bogBasketRotCtClockWiseMoveAllow.AppScalingDivisor :=1;
bogBasketRotCtClockWiseMoveAllow.AppScalingMultiplier :=1;
bogBasketRotCtClockWiseMoveAllow.AppScalingOffset :=0;
bogBasketRotCtClockWiseMoveAllow.AppUnit :="";
bogBasketRotCtClockWiseMoveAllow.CanDefault :=0;
bogBasketRotCtClockWiseMoveAllow.CanInit :=0;
bogBasketRotCtClockWiseMoveAllow.CanMax :=1;
bogBasketRotCtClockWiseMoveAllow.CanMin :=0;
bogBasketRotCtClockWiseMoveAllow.CanUnit :="";
bogBasketRotCtClockWiseMoveAllow.Description :="Basket Rotation Counter Clockwise Move Allowed";
bogBasketRotCtClockWiseMoveAllow.ErrorReaction := eErrorReaction.ERSIG_DFLT;
bogBasketRotCtClockWiseMoveAllow.ReceiverAdress :=1;
bogBasketRotCtClockWiseMoveAllow.ToolScalingDivisor :=1;
bogBasketRotCtClockWiseMoveAllow.ToolScalingMultiplier :=1;
bogBasketRotCtClockWiseMoveAllow.ToolScalingOffset :=0;
bogBasketRotCtClockWiseMoveAllow.ToolUnit :="";

bogBasketRotClockWiseMoveAllow.AppScalingDivisor :=1;
bogBasketRotClockWiseMoveAllow.AppScalingMultiplier :=1;
bogBasketRotClockWiseMoveAllow.AppScalingOffset :=0;
bogBasketRotClockWiseMoveAllow.AppUnit :="";
bogBasketRotClockWiseMoveAllow.CanDefault :=0;
bogBasketRotClockWiseMoveAllow.CanInit :=0;
bogBasketRotClockWiseMoveAllow.CanMax :=1;
bogBasketRotClockWiseMoveAllow.CanMin :=0;
bogBasketRotClockWiseMoveAllow.CanUnit :="";
bogBasketRotClockWiseMoveAllow.Description :="Basket Rotation Clockwise Move Allowed";
bogBasketRotClockWiseMoveAllow.ErrorReaction := eErrorReaction.ERSIG_DFLT;
bogBasketRotClockWiseMoveAllow.ReceiverAdress :=1;
bogBasketRotClockWiseMoveAllow.ToolScalingDivisor :=1;
bogBasketRotClockWiseMoveAllow.ToolScalingMultiplier :=1;
bogBasketRotClockWiseMoveAllow.ToolScalingOffset :=0;
bogBasketRotClockWiseMoveAllow.ToolUnit :="";

bogBasketInclinMoveUpAllow.AppScalingDivisor :=1;
bogBasketInclinMoveUpAllow.AppScalingMultiplier :=1;
bogBasketInclinMoveUpAllow.AppScalingOffset :=0;
bogBasketInclinMoveUpAllow.AppUnit :="";
bogBasketInclinMoveUpAllow.CanDefault :=0;
bogBasketInclinMoveUpAllow.CanInit :=0;
bogBasketInclinMoveUpAllow.CanMax :=1;
bogBasketInclinMoveUpAllow.CanMin :=0;
bogBasketInclinMoveUpAllow.CanUnit :="";
bogBasketInclinMoveUpAllow.Description :="Basket Inclinaison Move Up Allowed";
bogBasketInclinMoveUpAllow.ErrorReaction := eErrorReaction.ERSIG_DFLT;
bogBasketInclinMoveUpAllow.ReceiverAdress :=1;
bogBasketInclinMoveUpAllow.ToolScalingDivisor :=1;
bogBasketInclinMoveUpAllow.ToolScalingMultiplier :=1;
bogBasketInclinMoveUpAllow.ToolScalingOffset :=0;
bogBasketInclinMoveUpAllow.ToolUnit :="";

bogBasketInclinMoveDownAllow.AppScalingDivisor :=1;
bogBasketInclinMoveDownAllow.AppScalingMultiplier :=1;
bogBasketInclinMoveDownAllow.AppScalingOffset :=0;
bogBasketInclinMoveDownAllow.AppUnit :="";
bogBasketInclinMoveDownAllow.CanDefault :=0;
bogBasketInclinMoveDownAllow.CanInit :=0;
bogBasketInclinMoveDownAllow.CanMax :=1;
bogBasketInclinMoveDownAllow.CanMin :=0;
bogBasketInclinMoveDownAllow.CanUnit :="";
bogBasketInclinMoveDownAllow.Description :="Basket Inclinaison Move Down Allowed";
bogBasketInclinMoveDownAllow.ErrorReaction := eErrorReaction.ERSIG_DFLT;
bogBasketInclinMoveDownAllow.ReceiverAdress :=1;
bogBasketInclinMoveDownAllow.ToolScalingDivisor :=1;
bogBasketInclinMoveDownAllow.ToolScalingMultiplier :=1;
bogBasketInclinMoveDownAllow.ToolScalingOffset :=0;
bogBasketInclinMoveDownAllow.ToolUnit :="";

bogVehiculeDefault.AppScalingDivisor :=1;
bogVehiculeDefault.AppScalingMultiplier :=1;
bogVehiculeDefault.AppScalingOffset :=0;
bogVehiculeDefault.AppUnit :="";
bogVehiculeDefault.CanDefault :=0;
bogVehiculeDefault.CanInit :=0;
bogVehiculeDefault.CanMax :=1;
bogVehiculeDefault.CanMin :=0;
bogVehiculeDefault.CanUnit :="";
bogVehiculeDefault.Description :="Vehicule in Default (A12)";
bogVehiculeDefault.ErrorReaction := eErrorReaction.ERSIG_DFLT;
bogVehiculeDefault.ReceiverAdress :=1;
bogVehiculeDefault.ToolScalingDivisor :=1;
bogVehiculeDefault.ToolScalingMultiplier :=1;
bogVehiculeDefault.ToolScalingOffset :=0;
bogVehiculeDefault.ToolUnit :="";

bogTelescopeOutputPossible.AppScalingDivisor :=1;
bogTelescopeOutputPossible.AppScalingMultiplier :=1;
bogTelescopeOutputPossible.AppScalingOffset :=0;
bogTelescopeOutputPossible.AppUnit :="";
bogTelescopeOutputPossible.CanDefault :=0;
bogTelescopeOutputPossible.CanInit :=0;
bogTelescopeOutputPossible.CanMax :=1;
bogTelescopeOutputPossible.CanMin :=0;
bogTelescopeOutputPossible.CanUnit :="";
bogTelescopeOutputPossible.Description :="Telescope output possible (A48)";
bogTelescopeOutputPossible.ErrorReaction := eErrorReaction.ERSIG_DFLT;
bogTelescopeOutputPossible.ReceiverAdress :=1;
bogTelescopeOutputPossible.ToolScalingDivisor :=1;
bogTelescopeOutputPossible.ToolScalingMultiplier :=1;
bogTelescopeOutputPossible.ToolScalingOffset :=0;
bogTelescopeOutputPossible.ToolUnit :="";

bogTelescopeWinderFault.AppScalingDivisor :=1;
bogTelescopeWinderFault.AppScalingMultiplier :=1;
bogTelescopeWinderFault.AppScalingOffset :=0;
bogTelescopeWinderFault.AppUnit :="";
bogTelescopeWinderFault.CanDefault :=0;
bogTelescopeWinderFault.CanInit :=0;
bogTelescopeWinderFault.CanMax :=1;
bogTelescopeWinderFault.CanMin :=0;
bogTelescopeWinderFault.CanUnit :="";
bogTelescopeWinderFault.Description :="Telescope Winder Fault (A17)";
bogTelescopeWinderFault.ErrorReaction := eErrorReaction.ERSIG_DFLT;
bogTelescopeWinderFault.ReceiverAdress :=1;
bogTelescopeWinderFault.ToolScalingDivisor :=1;
bogTelescopeWinderFault.ToolScalingMultiplier :=1;
bogTelescopeWinderFault.ToolScalingOffset :=0;
bogTelescopeWinderFault.ToolUnit :="";

bogNacellePostSelector.AppScalingDivisor :=1;
bogNacellePostSelector.AppScalingMultiplier :=1;
bogNacellePostSelector.AppScalingOffset :=0;
bogNacellePostSelector.AppUnit :="";
bogNacellePostSelector.CanDefault :=0;
bogNacellePostSelector.CanInit :=0;
bogNacellePostSelector.CanMax :=1;
bogNacellePostSelector.CanMin :=0;
bogNacellePostSelector.CanUnit :="";
bogNacellePostSelector.Description :="Nacelle post selector";
bogNacellePostSelector.ErrorReaction := eErrorReaction.ERSIG_DFLT;
bogNacellePostSelector.ReceiverAdress :=1;
bogNacellePostSelector.ToolScalingDivisor :=1;
bogNacellePostSelector.ToolScalingMultiplier :=1;
bogNacellePostSelector.ToolScalingOffset :=0;
bogNacellePostSelector.ToolUnit :="";

bogSTOP_On_Off.AppScalingDivisor :=1;
bogSTOP_On_Off.AppScalingMultiplier :=1;
bogSTOP_On_Off.AppScalingOffset :=0;
bogSTOP_On_Off.AppUnit :="";
bogSTOP_On_Off.CanDefault :=0;
bogSTOP_On_Off.CanInit :=0;
bogSTOP_On_Off.CanMax :=1;
bogSTOP_On_Off.CanMin :=0;
bogSTOP_On_Off.CanUnit :="";
bogSTOP_On_Off.Description :="STOP Status";
bogSTOP_On_Off.ErrorReaction := eErrorReaction.ERSIG_DFLT;
bogSTOP_On_Off.ReceiverAdress :=1;
bogSTOP_On_Off.ToolScalingDivisor :=1;
bogSTOP_On_Off.ToolScalingMultiplier :=1;
bogSTOP_On_Off.ToolScalingOffset :=0;
bogSTOP_On_Off.ToolUnit :="";

bogSafeManSystem.AppScalingDivisor :=1;
bogSafeManSystem.AppScalingMultiplier :=1;
bogSafeManSystem.AppScalingOffset :=0;
bogSafeManSystem.AppUnit :="";
bogSafeManSystem.CanDefault :=0;
bogSafeManSystem.CanInit :=0;
bogSafeManSystem.CanMax :=1;
bogSafeManSystem.CanMin :=0;
bogSafeManSystem.CanUnit :="";
bogSafeManSystem.Description :="SafeManSystem (A5)";
bogSafeManSystem.ErrorReaction := eErrorReaction.ERSIG_DFLT;
bogSafeManSystem.ReceiverAdress :=1;
bogSafeManSystem.ToolScalingDivisor :=1;
bogSafeManSystem.ToolScalingMultiplier :=1;
bogSafeManSystem.ToolScalingOffset :=0;
bogSafeManSystem.ToolUnit :="";

bogHighSpeedAllow.AppScalingDivisor :=1;
bogHighSpeedAllow.AppScalingMultiplier :=1;
bogHighSpeedAllow.AppScalingOffset :=0;
bogHighSpeedAllow.AppUnit :="";
bogHighSpeedAllow.CanDefault :=0;
bogHighSpeedAllow.CanInit :=0;
bogHighSpeedAllow.CanMax :=1;
bogHighSpeedAllow.CanMin :=0;
bogHighSpeedAllow.CanUnit :="";
bogHighSpeedAllow.Description :="High Speed Allow (A19)";
bogHighSpeedAllow.ErrorReaction := eErrorReaction.ERSIG_DFLT;
bogHighSpeedAllow.ReceiverAdress :=1;
bogHighSpeedAllow.ToolScalingDivisor :=1;
bogHighSpeedAllow.ToolScalingMultiplier :=1;
bogHighSpeedAllow.ToolScalingOffset :=0;
bogHighSpeedAllow.ToolUnit :="";

bogAutomatiqueStop.AppScalingDivisor :=1;
bogAutomatiqueStop.AppScalingMultiplier :=1;
bogAutomatiqueStop.AppScalingOffset :=0;
bogAutomatiqueStop.AppUnit :="";
bogAutomatiqueStop.CanDefault :=0;
bogAutomatiqueStop.CanInit :=0;
bogAutomatiqueStop.CanMax :=1;
bogAutomatiqueStop.CanMin :=0;
bogAutomatiqueStop.CanUnit :="";
bogAutomatiqueStop.Description :="Automatique Stop or function mismatch (A20)";
bogAutomatiqueStop.ErrorReaction := eErrorReaction.ERSIG_DFLT;
bogAutomatiqueStop.ReceiverAdress :=1;
bogAutomatiqueStop.ToolScalingDivisor :=1;
bogAutomatiqueStop.ToolScalingMultiplier :=1;
bogAutomatiqueStop.ToolScalingOffset :=0;
bogAutomatiqueStop.ToolUnit :="";

bogLowSpeedByFault.AppScalingDivisor :=1;
bogLowSpeedByFault.AppScalingMultiplier :=1;
bogLowSpeedByFault.AppScalingOffset :=0;
bogLowSpeedByFault.AppUnit :="";
bogLowSpeedByFault.CanDefault :=0;
bogLowSpeedByFault.CanInit :=0;
bogLowSpeedByFault.CanMax :=1;
bogLowSpeedByFault.CanMin :=0;
bogLowSpeedByFault.CanUnit :="";
bogLowSpeedByFault.Description :="Low Speed by fault (A46)";
bogLowSpeedByFault.ErrorReaction := eErrorReaction.ERSIG_DFLT;
bogLowSpeedByFault.ReceiverAdress :=1;
bogLowSpeedByFault.ToolScalingDivisor :=1;
bogLowSpeedByFault.ToolScalingMultiplier :=1;
bogLowSpeedByFault.ToolScalingOffset :=0;
bogLowSpeedByFault.ToolUnit :="";

bogMeasuringMastFault.AppScalingDivisor :=1;
bogMeasuringMastFault.AppScalingMultiplier :=1;
bogMeasuringMastFault.AppScalingOffset :=0;
bogMeasuringMastFault.AppUnit :="";
bogMeasuringMastFault.CanDefault :=0;
bogMeasuringMastFault.CanInit :=0;
bogMeasuringMastFault.CanMax :=1;
bogMeasuringMastFault.CanMin :=0;
bogMeasuringMastFault.CanUnit :="";
bogMeasuringMastFault.Description :="Measuring Mast in Fault (A8)";
bogMeasuringMastFault.ErrorReaction := eErrorReaction.ERSIG_DFLT;
bogMeasuringMastFault.ReceiverAdress :=1;
bogMeasuringMastFault.ToolScalingDivisor :=1;
bogMeasuringMastFault.ToolScalingMultiplier :=1;
bogMeasuringMastFault.ToolScalingOffset :=0;
bogMeasuringMastFault.ToolUnit :="";

bogMeasuringMatOption.AppScalingDivisor :=1;
bogMeasuringMatOption.AppScalingMultiplier :=1;
bogMeasuringMatOption.AppScalingOffset :=0;
bogMeasuringMatOption.AppUnit :="";
bogMeasuringMatOption.CanDefault :=0;
bogMeasuringMatOption.CanInit :=0;
bogMeasuringMatOption.CanMax :=1;
bogMeasuringMatOption.CanMin :=0;
bogMeasuringMatOption.CanUnit :="";
bogMeasuringMatOption.Description :="Measuring mast option";
bogMeasuringMatOption.ErrorReaction := eErrorReaction.ERSIG_DFLT;
bogMeasuringMatOption.ReceiverAdress :=1;
bogMeasuringMatOption.ToolScalingDivisor :=1;
bogMeasuringMatOption.ToolScalingMultiplier :=1;
bogMeasuringMatOption.ToolScalingOffset :=0;
bogMeasuringMatOption.ToolUnit :="";

bogBasketAccessLocked.AppScalingDivisor :=1;
bogBasketAccessLocked.AppScalingMultiplier :=1;
bogBasketAccessLocked.AppScalingOffset :=0;
bogBasketAccessLocked.AppUnit :="";
bogBasketAccessLocked.CanDefault :=0;
bogBasketAccessLocked.CanInit :=0;
bogBasketAccessLocked.CanMax :=1;
bogBasketAccessLocked.CanMin :=0;
bogBasketAccessLocked.CanUnit :="";
bogBasketAccessLocked.Description :="Basket access locked";
bogBasketAccessLocked.ErrorReaction := eErrorReaction.ERSIG_DFLT;
bogBasketAccessLocked.ReceiverAdress :=1;
bogBasketAccessLocked.ToolScalingDivisor :=1;
bogBasketAccessLocked.ToolScalingMultiplier :=1;
bogBasketAccessLocked.ToolScalingOffset :=0;
bogBasketAccessLocked.ToolUnit :="";

bogFilterOverloadNoActive.AppScalingDivisor :=1;
bogFilterOverloadNoActive.AppScalingMultiplier :=1;
bogFilterOverloadNoActive.AppScalingOffset :=0;
bogFilterOverloadNoActive.AppUnit :="";
bogFilterOverloadNoActive.CanDefault :=0;
bogFilterOverloadNoActive.CanInit :=0;
bogFilterOverloadNoActive.CanMax :=1;
bogFilterOverloadNoActive.CanMin :=0;
bogFilterOverloadNoActive.CanUnit :="";
bogFilterOverloadNoActive.Description :="new signal";
bogFilterOverloadNoActive.ErrorReaction := eErrorReaction.ERSIG_DFLT;
bogFilterOverloadNoActive.ReceiverAdress :=1;
bogFilterOverloadNoActive.ToolScalingDivisor :=1;
bogFilterOverloadNoActive.ToolScalingMultiplier :=1;
bogFilterOverloadNoActive.ToolScalingOffset :=0;
bogFilterOverloadNoActive.ToolUnit :="";

bogAnticlockwiseBasketSlew.AppScalingDivisor :=1;
bogAnticlockwiseBasketSlew.AppScalingMultiplier :=1;
bogAnticlockwiseBasketSlew.AppScalingOffset :=0;
bogAnticlockwiseBasketSlew.AppUnit :="";
bogAnticlockwiseBasketSlew.CanDefault :=0;
bogAnticlockwiseBasketSlew.CanInit :=0;
bogAnticlockwiseBasketSlew.CanMax :=1;
bogAnticlockwiseBasketSlew.CanMin :=0;
bogAnticlockwiseBasketSlew.CanUnit :="";
bogAnticlockwiseBasketSlew.Description :="EV113 Anticlockwise Basket Slew";
bogAnticlockwiseBasketSlew.ErrorReaction := eErrorReaction.ERSIG_DFLT;
bogAnticlockwiseBasketSlew.ReceiverAdress :=1;
bogAnticlockwiseBasketSlew.ToolScalingDivisor :=1;
bogAnticlockwiseBasketSlew.ToolScalingMultiplier :=1;
bogAnticlockwiseBasketSlew.ToolScalingOffset :=0;
bogAnticlockwiseBasketSlew.ToolUnit :="";

bogClockwiseBasketSlew.AppScalingDivisor :=1;
bogClockwiseBasketSlew.AppScalingMultiplier :=1;
bogClockwiseBasketSlew.AppScalingOffset :=0;
bogClockwiseBasketSlew.AppUnit :="";
bogClockwiseBasketSlew.CanDefault :=0;
bogClockwiseBasketSlew.CanInit :=0;
bogClockwiseBasketSlew.CanMax :=1;
bogClockwiseBasketSlew.CanMin :=0;
bogClockwiseBasketSlew.CanUnit :="";
bogClockwiseBasketSlew.Description :="EV112 Anticlockwise Basket Slew";
bogClockwiseBasketSlew.ErrorReaction := eErrorReaction.ERSIG_DFLT;
bogClockwiseBasketSlew.ReceiverAdress :=1;
bogClockwiseBasketSlew.ToolScalingDivisor :=1;
bogClockwiseBasketSlew.ToolScalingMultiplier :=1;
bogClockwiseBasketSlew.ToolScalingOffset :=0;
bogClockwiseBasketSlew.ToolUnit :="";

bogFlashLightForced.AppScalingDivisor :=1;
bogFlashLightForced.AppScalingMultiplier :=1;
bogFlashLightForced.AppScalingOffset :=0;
bogFlashLightForced.AppUnit :="";
bogFlashLightForced.CanDefault :=0;
bogFlashLightForced.CanInit :=0;
bogFlashLightForced.CanMax :=1;
bogFlashLightForced.CanMin :=0;
bogFlashLightForced.CanUnit :="";
bogFlashLightForced.Description :="Flash Light Forced";
bogFlashLightForced.ErrorReaction := eErrorReaction.ERSIG_DFLT;
bogFlashLightForced.ReceiverAdress :=1;
bogFlashLightForced.ToolScalingDivisor :=1;
bogFlashLightForced.ToolScalingMultiplier :=1;
bogFlashLightForced.ToolScalingOffset :=0;
bogFlashLightForced.ToolUnit :="";

bogBasketAccessLockOption.AppScalingDivisor :=1;
bogBasketAccessLockOption.AppScalingMultiplier :=1;
bogBasketAccessLockOption.AppScalingOffset :=0;
bogBasketAccessLockOption.AppUnit :="";
bogBasketAccessLockOption.CanDefault :=0;
bogBasketAccessLockOption.CanInit :=0;
bogBasketAccessLockOption.CanMax :=1;
bogBasketAccessLockOption.CanMin :=0;
bogBasketAccessLockOption.CanUnit :="";
bogBasketAccessLockOption.Description :="Basket Lock Option";
bogBasketAccessLockOption.ErrorReaction := eErrorReaction.ERSIG_DFLT;
bogBasketAccessLockOption.ReceiverAdress :=1;
bogBasketAccessLockOption.ToolScalingDivisor :=1;
bogBasketAccessLockOption.ToolScalingMultiplier :=1;
bogBasketAccessLockOption.ToolScalingOffset :=0;
bogBasketAccessLockOption.ToolUnit :="";

bogBasketLateralStopOption.AppScalingDivisor :=1;
bogBasketLateralStopOption.AppScalingMultiplier :=1;
bogBasketLateralStopOption.AppScalingOffset :=0;
bogBasketLateralStopOption.AppUnit :="";
bogBasketLateralStopOption.CanDefault :=0;
bogBasketLateralStopOption.CanInit :=0;
bogBasketLateralStopOption.CanMax :=1;
bogBasketLateralStopOption.CanMin :=0;
bogBasketLateralStopOption.CanUnit :="";
bogBasketLateralStopOption.Description :="Basket lateral stop option";
bogBasketLateralStopOption.ErrorReaction := eErrorReaction.ERSIG_DFLT;
bogBasketLateralStopOption.ReceiverAdress :=1;
bogBasketLateralStopOption.ToolScalingDivisor :=1;
bogBasketLateralStopOption.ToolScalingMultiplier :=1;
bogBasketLateralStopOption.ToolScalingOffset :=0;
bogBasketLateralStopOption.ToolUnit :="";

bogBasketStepClosed.AppScalingDivisor :=1;
bogBasketStepClosed.AppScalingMultiplier :=1;
bogBasketStepClosed.AppScalingOffset :=0;
bogBasketStepClosed.AppUnit :="";
bogBasketStepClosed.CanDefault :=0;
bogBasketStepClosed.CanInit :=0;
bogBasketStepClosed.CanMax :=1;
bogBasketStepClosed.CanMin :=0;
bogBasketStepClosed.CanUnit :="";
bogBasketStepClosed.Description :="Basket step closed";
bogBasketStepClosed.ErrorReaction := eErrorReaction.ERSIG_DFLT;
bogBasketStepClosed.ReceiverAdress :=1;
bogBasketStepClosed.ToolScalingDivisor :=1;
bogBasketStepClosed.ToolScalingMultiplier :=1;
bogBasketStepClosed.ToolScalingOffset :=0;
bogBasketStepClosed.ToolUnit :="";

bogSystemFault.AppScalingDivisor :=1;
bogSystemFault.AppScalingMultiplier :=1;
bogSystemFault.AppScalingOffset :=0;
bogSystemFault.AppUnit :="";
bogSystemFault.CanDefault :=0;
bogSystemFault.CanInit :=0;
bogSystemFault.CanMax :=1;
bogSystemFault.CanMin :=0;
bogSystemFault.CanUnit :="";
bogSystemFault.Description :="System Fault";
bogSystemFault.ErrorReaction := eErrorReaction.ERSIG_DFLT;
bogSystemFault.ReceiverAdress :=1;
bogSystemFault.ToolScalingDivisor :=1;
bogSystemFault.ToolScalingMultiplier :=1;
bogSystemFault.ToolScalingOffset :=0;
bogSystemFault.ToolUnit :="";

bogTrans1PressureSensorFault.AppScalingDivisor :=1;
bogTrans1PressureSensorFault.AppScalingMultiplier :=1;
bogTrans1PressureSensorFault.AppScalingOffset :=0;
bogTrans1PressureSensorFault.AppUnit :="";
bogTrans1PressureSensorFault.CanDefault :=0;
bogTrans1PressureSensorFault.CanInit :=0;
bogTrans1PressureSensorFault.CanMax :=1;
bogTrans1PressureSensorFault.CanMin :=0;
bogTrans1PressureSensorFault.CanUnit :="";
bogTrans1PressureSensorFault.Description :="Fault pressure transmission 1";
bogTrans1PressureSensorFault.ErrorReaction := eErrorReaction.ERSIG_DFLT;
bogTrans1PressureSensorFault.ReceiverAdress :=1;
bogTrans1PressureSensorFault.ToolScalingDivisor :=1;
bogTrans1PressureSensorFault.ToolScalingMultiplier :=1;
bogTrans1PressureSensorFault.ToolScalingOffset :=0;
bogTrans1PressureSensorFault.ToolUnit :="";

bogTrans2PressureSensorFault.AppScalingDivisor :=1;
bogTrans2PressureSensorFault.AppScalingMultiplier :=1;
bogTrans2PressureSensorFault.AppScalingOffset :=0;
bogTrans2PressureSensorFault.AppUnit :="";
bogTrans2PressureSensorFault.CanDefault :=0;
bogTrans2PressureSensorFault.CanInit :=0;
bogTrans2PressureSensorFault.CanMax :=1;
bogTrans2PressureSensorFault.CanMin :=0;
bogTrans2PressureSensorFault.CanUnit :="";
bogTrans2PressureSensorFault.Description :="Fault pressure transmission 2";
bogTrans2PressureSensorFault.ErrorReaction := eErrorReaction.ERSIG_DFLT;
bogTrans2PressureSensorFault.ReceiverAdress :=1;
bogTrans2PressureSensorFault.ToolScalingDivisor :=1;
bogTrans2PressureSensorFault.ToolScalingMultiplier :=1;
bogTrans2PressureSensorFault.ToolScalingOffset :=0;
bogTrans2PressureSensorFault.ToolUnit :="";

bogOverloadSecurity.AppScalingDivisor :=1;
bogOverloadSecurity.AppScalingMultiplier :=1;
bogOverloadSecurity.AppScalingOffset :=0;
bogOverloadSecurity.AppUnit :="";
bogOverloadSecurity.CanDefault :=0;
bogOverloadSecurity.CanInit :=0;
bogOverloadSecurity.CanMax :=1;
bogOverloadSecurity.CanMin :=0;
bogOverloadSecurity.CanUnit :="";
bogOverloadSecurity.Description :="Basket overload";
bogOverloadSecurity.ErrorReaction := eErrorReaction.ERSIG_DFLT;
bogOverloadSecurity.ReceiverAdress :=1;
bogOverloadSecurity.ToolScalingDivisor :=1;
bogOverloadSecurity.ToolScalingMultiplier :=1;
bogOverloadSecurity.ToolScalingOffset :=0;
bogOverloadSecurity.ToolUnit :="";

bogDeltaArmJoysCenteredTeles.AppScalingDivisor :=1;
bogDeltaArmJoysCenteredTeles.AppScalingMultiplier :=1;
bogDeltaArmJoysCenteredTeles.AppScalingOffset :=0;
bogDeltaArmJoysCenteredTeles.AppUnit :="";
bogDeltaArmJoysCenteredTeles.CanDefault :=0;
bogDeltaArmJoysCenteredTeles.CanInit :=0;
bogDeltaArmJoysCenteredTeles.CanMax :=1;
bogDeltaArmJoysCenteredTeles.CanMin :=0;
bogDeltaArmJoysCenteredTeles.CanUnit :="";
bogDeltaArmJoysCenteredTeles.Description :="Delta and Telescope Joystick centered";
bogDeltaArmJoysCenteredTeles.ErrorReaction := eErrorReaction.ERSIG_DFLT;
bogDeltaArmJoysCenteredTeles.ReceiverAdress :=1;
bogDeltaArmJoysCenteredTeles.ToolScalingDivisor :=1;
bogDeltaArmJoysCenteredTeles.ToolScalingMultiplier :=1;
bogDeltaArmJoysCenteredTeles.ToolScalingOffset :=0;
bogDeltaArmJoysCenteredTeles.ToolUnit :="";

bogArrowJoystickCenteredTurret.AppScalingDivisor :=1;
bogArrowJoystickCenteredTurret.AppScalingMultiplier :=1;
bogArrowJoystickCenteredTurret.AppScalingOffset :=0;
bogArrowJoystickCenteredTurret.AppUnit :="";
bogArrowJoystickCenteredTurret.CanDefault :=0;
bogArrowJoystickCenteredTurret.CanInit :=0;
bogArrowJoystickCenteredTurret.CanMax :=1;
bogArrowJoystickCenteredTurret.CanMin :=0;
bogArrowJoystickCenteredTurret.CanUnit :="";
bogArrowJoystickCenteredTurret.Description :="Arrow and Turret Joystick centered";
bogArrowJoystickCenteredTurret.ErrorReaction := eErrorReaction.ERSIG_DFLT;
bogArrowJoystickCenteredTurret.ReceiverAdress :=1;
bogArrowJoystickCenteredTurret.ToolScalingDivisor :=1;
bogArrowJoystickCenteredTurret.ToolScalingMultiplier :=1;
bogArrowJoystickCenteredTurret.ToolScalingOffset :=0;
bogArrowJoystickCenteredTurret.ToolUnit :="";

bogDeltaArmMoveUp.AppScalingDivisor :=1;
bogDeltaArmMoveUp.AppScalingMultiplier :=1;
bogDeltaArmMoveUp.AppScalingOffset :=0;
bogDeltaArmMoveUp.AppUnit :="";
bogDeltaArmMoveUp.CanDefault :=0;
bogDeltaArmMoveUp.CanInit :=0;
bogDeltaArmMoveUp.CanMax :=1;
bogDeltaArmMoveUp.CanMin :=0;
bogDeltaArmMoveUp.CanUnit :="";
bogDeltaArmMoveUp.Description :="Delta Arm Move Up";
bogDeltaArmMoveUp.ErrorReaction := eErrorReaction.ERSIG_DFLT;
bogDeltaArmMoveUp.ReceiverAdress :=1;
bogDeltaArmMoveUp.ToolScalingDivisor :=1;
bogDeltaArmMoveUp.ToolScalingMultiplier :=1;
bogDeltaArmMoveUp.ToolScalingOffset :=0;
bogDeltaArmMoveUp.ToolUnit :="";

bogDeltaArmMoveDown.AppScalingDivisor :=1;
bogDeltaArmMoveDown.AppScalingMultiplier :=1;
bogDeltaArmMoveDown.AppScalingOffset :=0;
bogDeltaArmMoveDown.AppUnit :="";
bogDeltaArmMoveDown.CanDefault :=0;
bogDeltaArmMoveDown.CanInit :=0;
bogDeltaArmMoveDown.CanMax :=1;
bogDeltaArmMoveDown.CanMin :=0;
bogDeltaArmMoveDown.CanUnit :="";
bogDeltaArmMoveDown.Description :="Delta Arm Move Down";
bogDeltaArmMoveDown.ErrorReaction := eErrorReaction.ERSIG_DFLT;
bogDeltaArmMoveDown.ReceiverAdress :=1;
bogDeltaArmMoveDown.ToolScalingDivisor :=1;
bogDeltaArmMoveDown.ToolScalingMultiplier :=1;
bogDeltaArmMoveDown.ToolScalingOffset :=0;
bogDeltaArmMoveDown.ToolUnit :="";

bogArrowArmMoveUp.AppScalingDivisor :=1;
bogArrowArmMoveUp.AppScalingMultiplier :=1;
bogArrowArmMoveUp.AppScalingOffset :=0;
bogArrowArmMoveUp.AppUnit :="";
bogArrowArmMoveUp.CanDefault :=0;
bogArrowArmMoveUp.CanInit :=0;
bogArrowArmMoveUp.CanMax :=1;
bogArrowArmMoveUp.CanMin :=0;
bogArrowArmMoveUp.CanUnit :="";
bogArrowArmMoveUp.Description :="Arrow Arm Move Up";
bogArrowArmMoveUp.ErrorReaction := eErrorReaction.ERSIG_DFLT;
bogArrowArmMoveUp.ReceiverAdress :=1;
bogArrowArmMoveUp.ToolScalingDivisor :=1;
bogArrowArmMoveUp.ToolScalingMultiplier :=1;
bogArrowArmMoveUp.ToolScalingOffset :=0;
bogArrowArmMoveUp.ToolUnit :="";

bogArrowArmMoveDown.AppScalingDivisor :=1;
bogArrowArmMoveDown.AppScalingMultiplier :=1;
bogArrowArmMoveDown.AppScalingOffset :=0;
bogArrowArmMoveDown.AppUnit :="";
bogArrowArmMoveDown.CanDefault :=0;
bogArrowArmMoveDown.CanInit :=0;
bogArrowArmMoveDown.CanMax :=1;
bogArrowArmMoveDown.CanMin :=0;
bogArrowArmMoveDown.CanUnit :="";
bogArrowArmMoveDown.Description :="Arrow Arm Move Down";
bogArrowArmMoveDown.ErrorReaction := eErrorReaction.ERSIG_DFLT;
bogArrowArmMoveDown.ReceiverAdress :=1;
bogArrowArmMoveDown.ToolScalingDivisor :=1;
bogArrowArmMoveDown.ToolScalingMultiplier :=1;
bogArrowArmMoveDown.ToolScalingOffset :=0;
bogArrowArmMoveDown.ToolUnit :="";

bogTelescopeMoveOut.AppScalingDivisor :=1;
bogTelescopeMoveOut.AppScalingMultiplier :=1;
bogTelescopeMoveOut.AppScalingOffset :=0;
bogTelescopeMoveOut.AppUnit :="";
bogTelescopeMoveOut.CanDefault :=0;
bogTelescopeMoveOut.CanInit :=0;
bogTelescopeMoveOut.CanMax :=1;
bogTelescopeMoveOut.CanMin :=0;
bogTelescopeMoveOut.CanUnit :="";
bogTelescopeMoveOut.Description :="Telescope Move Out";
bogTelescopeMoveOut.ErrorReaction := eErrorReaction.ERSIG_DFLT;
bogTelescopeMoveOut.ReceiverAdress :=1;
bogTelescopeMoveOut.ToolScalingDivisor :=1;
bogTelescopeMoveOut.ToolScalingMultiplier :=1;
bogTelescopeMoveOut.ToolScalingOffset :=0;
bogTelescopeMoveOut.ToolUnit :="";

bogTelescopeMoveIn.AppScalingDivisor :=1;
bogTelescopeMoveIn.AppScalingMultiplier :=1;
bogTelescopeMoveIn.AppScalingOffset :=0;
bogTelescopeMoveIn.AppUnit :="";
bogTelescopeMoveIn.CanDefault :=0;
bogTelescopeMoveIn.CanInit :=0;
bogTelescopeMoveIn.CanMax :=1;
bogTelescopeMoveIn.CanMin :=0;
bogTelescopeMoveIn.CanUnit :="";
bogTelescopeMoveIn.Description :="Telescope Move In";
bogTelescopeMoveIn.ErrorReaction := eErrorReaction.ERSIG_DFLT;
bogTelescopeMoveIn.ReceiverAdress :=1;
bogTelescopeMoveIn.ToolScalingDivisor :=1;
bogTelescopeMoveIn.ToolScalingMultiplier :=1;
bogTelescopeMoveIn.ToolScalingOffset :=0;
bogTelescopeMoveIn.ToolUnit :="";

bogTurretCounterClockWiseMove.AppScalingDivisor :=1;
bogTurretCounterClockWiseMove.AppScalingMultiplier :=1;
bogTurretCounterClockWiseMove.AppScalingOffset :=0;
bogTurretCounterClockWiseMove.AppUnit :="";
bogTurretCounterClockWiseMove.CanDefault :=0;
bogTurretCounterClockWiseMove.CanInit :=0;
bogTurretCounterClockWiseMove.CanMax :=1;
bogTurretCounterClockWiseMove.CanMin :=0;
bogTurretCounterClockWiseMove.CanUnit :="";
bogTurretCounterClockWiseMove.Description :="Turret Counter Clockwise Move";
bogTurretCounterClockWiseMove.ErrorReaction := eErrorReaction.ERSIG_DFLT;
bogTurretCounterClockWiseMove.ReceiverAdress :=1;
bogTurretCounterClockWiseMove.ToolScalingDivisor :=1;
bogTurretCounterClockWiseMove.ToolScalingMultiplier :=1;
bogTurretCounterClockWiseMove.ToolScalingOffset :=0;
bogTurretCounterClockWiseMove.ToolUnit :="";

bogTurretClockWiseMove.AppScalingDivisor :=1;
bogTurretClockWiseMove.AppScalingMultiplier :=1;
bogTurretClockWiseMove.AppScalingOffset :=0;
bogTurretClockWiseMove.AppUnit :="";
bogTurretClockWiseMove.CanDefault :=0;
bogTurretClockWiseMove.CanInit :=0;
bogTurretClockWiseMove.CanMax :=1;
bogTurretClockWiseMove.CanMin :=0;
bogTurretClockWiseMove.CanUnit :="";
bogTurretClockWiseMove.Description :="Turret Clockwise Move";
bogTurretClockWiseMove.ErrorReaction := eErrorReaction.ERSIG_DFLT;
bogTurretClockWiseMove.ReceiverAdress :=1;
bogTurretClockWiseMove.ToolScalingDivisor :=1;
bogTurretClockWiseMove.ToolScalingMultiplier :=1;
bogTurretClockWiseMove.ToolScalingOffset :=0;
bogTurretClockWiseMove.ToolUnit :="";

bogTurretEncoderFault.AppScalingDivisor :=1;
bogTurretEncoderFault.AppScalingMultiplier :=1;
bogTurretEncoderFault.AppScalingOffset :=0;
bogTurretEncoderFault.AppUnit :="";
bogTurretEncoderFault.CanDefault :=0;
bogTurretEncoderFault.CanInit :=0;
bogTurretEncoderFault.CanMax :=1;
bogTurretEncoderFault.CanMin :=0;
bogTurretEncoderFault.CanUnit :="";
bogTurretEncoderFault.Description :="Turret Encoder Fault";
bogTurretEncoderFault.ErrorReaction := eErrorReaction.ERSIG_DFLT;
bogTurretEncoderFault.ReceiverAdress :=1;
bogTurretEncoderFault.ToolScalingDivisor :=1;
bogTurretEncoderFault.ToolScalingMultiplier :=1;
bogTurretEncoderFault.ToolScalingOffset :=0;
bogTurretEncoderFault.ToolUnit :="";

bogGeneratorOption.AppScalingDivisor :=1;
bogGeneratorOption.AppScalingMultiplier :=1;
bogGeneratorOption.AppScalingOffset :=0;
bogGeneratorOption.AppUnit :="";
bogGeneratorOption.CanDefault :=0;
bogGeneratorOption.CanInit :=0;
bogGeneratorOption.CanMax :=1;
bogGeneratorOption.CanMin :=0;
bogGeneratorOption.CanUnit :="";
bogGeneratorOption.Description :="Generator Option";
bogGeneratorOption.ErrorReaction := eErrorReaction.ERSIG_DFLT;
bogGeneratorOption.ReceiverAdress :=1;
bogGeneratorOption.ToolScalingDivisor :=1;
bogGeneratorOption.ToolScalingMultiplier :=1;
bogGeneratorOption.ToolScalingOffset :=0;
bogGeneratorOption.ToolUnit :="";

bogGeneratorActive.AppScalingDivisor :=1;
bogGeneratorActive.AppScalingMultiplier :=1;
bogGeneratorActive.AppScalingOffset :=0;
bogGeneratorActive.AppUnit :="";
bogGeneratorActive.CanDefault :=0;
bogGeneratorActive.CanInit :=0;
bogGeneratorActive.CanMax :=1;
bogGeneratorActive.CanMin :=0;
bogGeneratorActive.CanUnit :="";
bogGeneratorActive.Description :="Generator Active";
bogGeneratorActive.ErrorReaction := eErrorReaction.ERSIG_DFLT;
bogGeneratorActive.ReceiverAdress :=1;
bogGeneratorActive.ToolScalingDivisor :=1;
bogGeneratorActive.ToolScalingMultiplier :=1;
bogGeneratorActive.ToolScalingOffset :=0;
bogGeneratorActive.ToolUnit :="";


                
END_METHOD
END_FUNCTION_BLOCK

FUNCTION_BLOCK Msg2C1SendToEvision7MessageClass EXTENDS CanReceiveMessageClass
  VAR_INPUT
    u8gFuel : UInt8CanSignalClass;
    u16gBattery_Voltage : UInt16CanSignalClass;
    u8gTrainTransmissionPressure : UInt8CanSignalClass;
    i16gBypassPressureSensorValue : Int16CanSignalClass;
    Counter : UInt32CanSignalClass;
  END_VAR

            
          

METHOD SetData
  VAR_INPUT
    CanMsgPointer : POINTER TO CanMessageClass;
  END_VAR
                  IF IsValidPointer(canMsgPointer,'SetData') THEN
	SUPER^.SetData(CanMsgPointer);
	//Set the new data
	u8gFuel.Value := canMsgPointer^.GetUint8(0);
	u16gBattery_Voltage.Value := canMsgPointer^.GetUint16(8);
	u8gTrainTransmissionPressure.Value := canMsgPointer^.GetUint8(24);
	i16gBypassPressureSensorValue.Value := canMsgPointer^.GetInt16(32);
	//And increase the counter
	Counter.Value := CanMsgPointer^.Counter.Value;
END_IF

                
END_METHOD

PROPERTY u8gFuelRawValue : USINT
GET
                    IF u8gFuel.AppScalingMultiplier = 0 THEN
	_MatchLog^.Error("Get u8gFuelRawValue", "Division by Zero!");
	RETURN;
End_IF

u8gFuelRawValue := TO_USINT((u8gFuel.Value - u8gFuel.AppScalingOffset) * u8gFuel.AppScalingDivisor / u8gFuel.AppScalingMultiplier);

                  
END_GET
END_PROPERTY

PROPERTY u16gBattery_VoltageRawValue : UINT
GET
                    IF u16gBattery_Voltage.AppScalingMultiplier = 0 THEN
	_MatchLog^.Error("Get u16gBattery_VoltageRawValue", "Division by Zero!");
	RETURN;
End_IF

u16gBattery_VoltageRawValue := TO_UINT((u16gBattery_Voltage.Value - u16gBattery_Voltage.AppScalingOffset) * u16gBattery_Voltage.AppScalingDivisor / u16gBattery_Voltage.AppScalingMultiplier);

                  
END_GET
END_PROPERTY

PROPERTY u8gTrainTransmissionPressureRawValue : USINT
GET
                    IF u8gTrainTransmissionPressure.AppScalingMultiplier = 0 THEN
	_MatchLog^.Error("Get u8gTrainTransmissionPressureRawValue", "Division by Zero!");
	RETURN;
End_IF

u8gTrainTransmissionPressureRawValue := TO_USINT((u8gTrainTransmissionPressure.Value - u8gTrainTransmissionPressure.AppScalingOffset) * u8gTrainTransmissionPressure.AppScalingDivisor / u8gTrainTransmissionPressure.AppScalingMultiplier);

                  
END_GET
END_PROPERTY

PROPERTY i16gBypassPressureSensorValueRawValue : INT
GET
                    IF i16gBypassPressureSensorValue.AppScalingMultiplier = 0 THEN
	_MatchLog^.Error("Get i16gBypassPressureSensorValueRawValue", "Division by Zero!");
	RETURN;
End_IF

i16gBypassPressureSensorValueRawValue := TO_INT((i16gBypassPressureSensorValue.Value - i16gBypassPressureSensorValue.AppScalingOffset) * i16gBypassPressureSensorValue.AppScalingDivisor / i16gBypassPressureSensorValue.AppScalingMultiplier);

                  
END_GET
END_PROPERTY

PROPERTY u8gFuelToolValue : USINT
GET
                    IF u8gFuel.ToolScalingDivisor = 0 OR u8gFuel.AppScalingMultiplier = 0 THEN
	_MatchLog^.Error("Get u8gFuelToolValue", "Division by Zero!");
	RETURN;
END_IF

u8gFuelToolValue := TO_USINT(((u8gFuel.Value - u8gFuel.AppScalingOffset) * u8gFuel.AppScalingDivisor / u8gFuel.AppScalingMultiplier * u8gFuel.ToolScalingMultiplier / u8gFuel.ToolScalingDivisor) + u8gFuel.ToolScalingOffset);

                  
END_GET
END_PROPERTY

PROPERTY u16gBattery_VoltageToolValue : UINT
GET
                    IF u16gBattery_Voltage.ToolScalingDivisor = 0 OR u16gBattery_Voltage.AppScalingMultiplier = 0 THEN
	_MatchLog^.Error("Get u16gBattery_VoltageToolValue", "Division by Zero!");
	RETURN;
END_IF

u16gBattery_VoltageToolValue := TO_UINT(((u16gBattery_Voltage.Value - u16gBattery_Voltage.AppScalingOffset) * u16gBattery_Voltage.AppScalingDivisor / u16gBattery_Voltage.AppScalingMultiplier * u16gBattery_Voltage.ToolScalingMultiplier / u16gBattery_Voltage.ToolScalingDivisor) + u16gBattery_Voltage.ToolScalingOffset);

                  
END_GET
END_PROPERTY

PROPERTY u8gTrainTransmissionPressureToolValue : USINT
GET
                    IF u8gTrainTransmissionPressure.ToolScalingDivisor = 0 OR u8gTrainTransmissionPressure.AppScalingMultiplier = 0 THEN
	_MatchLog^.Error("Get u8gTrainTransmissionPressureToolValue", "Division by Zero!");
	RETURN;
END_IF

u8gTrainTransmissionPressureToolValue := TO_USINT(((u8gTrainTransmissionPressure.Value - u8gTrainTransmissionPressure.AppScalingOffset) * u8gTrainTransmissionPressure.AppScalingDivisor / u8gTrainTransmissionPressure.AppScalingMultiplier * u8gTrainTransmissionPressure.ToolScalingMultiplier / u8gTrainTransmissionPressure.ToolScalingDivisor) + u8gTrainTransmissionPressure.ToolScalingOffset);

                  
END_GET
END_PROPERTY

PROPERTY i16gBypassPressureSensorValueToolValue : INT
GET
                    IF i16gBypassPressureSensorValue.ToolScalingDivisor = 0 OR i16gBypassPressureSensorValue.AppScalingMultiplier = 0 THEN
	_MatchLog^.Error("Get i16gBypassPressureSensorValueToolValue", "Division by Zero!");
	RETURN;
END_IF

i16gBypassPressureSensorValueToolValue := TO_INT(((i16gBypassPressureSensorValue.Value - i16gBypassPressureSensorValue.AppScalingOffset) * i16gBypassPressureSensorValue.AppScalingDivisor / i16gBypassPressureSensorValue.AppScalingMultiplier * i16gBypassPressureSensorValue.ToolScalingMultiplier / i16gBypassPressureSensorValue.ToolScalingDivisor) + i16gBypassPressureSensorValue.ToolScalingOffset);

                  
END_GET
END_PROPERTY

METHOD InitializeCanSignals
                  u8gFuel.AppScalingDivisor :=1;
u8gFuel.AppScalingMultiplier :=1;
u8gFuel.AppScalingOffset :=0;
u8gFuel.AppUnit :="";
u8gFuel.CanDefault :=0;
u8gFuel.CanInit :=0;
u8gFuel.CanMax :=255;
u8gFuel.CanMin :=0;
u8gFuel.CanUnit :="";
u8gFuel.Description :="new signal";
u8gFuel.ErrorReaction := eErrorReaction.ERSIG_DFLT;
u8gFuel.ReceiverAdress :=1;
u8gFuel.ToolScalingDivisor :=1;
u8gFuel.ToolScalingMultiplier :=1;
u8gFuel.ToolScalingOffset :=0;
u8gFuel.ToolUnit :="";

u16gBattery_Voltage.AppScalingDivisor :=1;
u16gBattery_Voltage.AppScalingMultiplier :=1;
u16gBattery_Voltage.AppScalingOffset :=0;
u16gBattery_Voltage.AppUnit :="";
u16gBattery_Voltage.CanDefault :=0;
u16gBattery_Voltage.CanInit :=0;
u16gBattery_Voltage.CanMax :=65535;
u16gBattery_Voltage.CanMin :=0;
u16gBattery_Voltage.CanUnit :="";
u16gBattery_Voltage.Description :="new signal";
u16gBattery_Voltage.ErrorReaction := eErrorReaction.ERSIG_DFLT;
u16gBattery_Voltage.ReceiverAdress :=1;
u16gBattery_Voltage.ToolScalingDivisor :=1;
u16gBattery_Voltage.ToolScalingMultiplier :=1;
u16gBattery_Voltage.ToolScalingOffset :=0;
u16gBattery_Voltage.ToolUnit :="";

u8gTrainTransmissionPressure.AppScalingDivisor :=1;
u8gTrainTransmissionPressure.AppScalingMultiplier :=1;
u8gTrainTransmissionPressure.AppScalingOffset :=0;
u8gTrainTransmissionPressure.AppUnit :="";
u8gTrainTransmissionPressure.CanDefault :=0;
u8gTrainTransmissionPressure.CanInit :=0;
u8gTrainTransmissionPressure.CanMax :=255;
u8gTrainTransmissionPressure.CanMin :=0;
u8gTrainTransmissionPressure.CanUnit :="";
u8gTrainTransmissionPressure.Description :="new signal";
u8gTrainTransmissionPressure.ErrorReaction := eErrorReaction.ERSIG_DFLT;
u8gTrainTransmissionPressure.ReceiverAdress :=1;
u8gTrainTransmissionPressure.ToolScalingDivisor :=1;
u8gTrainTransmissionPressure.ToolScalingMultiplier :=1;
u8gTrainTransmissionPressure.ToolScalingOffset :=0;
u8gTrainTransmissionPressure.ToolUnit :="";

i16gBypassPressureSensorValue.AppScalingDivisor :=1;
i16gBypassPressureSensorValue.AppScalingMultiplier :=1;
i16gBypassPressureSensorValue.AppScalingOffset :=0;
i16gBypassPressureSensorValue.AppUnit :="";
i16gBypassPressureSensorValue.CanDefault :=0;
i16gBypassPressureSensorValue.CanInit :=0;
i16gBypassPressureSensorValue.CanMax :=VBasic.LibConst.I16_MAX;
i16gBypassPressureSensorValue.CanMin :=VBasic.LibConst.I16_MIN;
i16gBypassPressureSensorValue.CanUnit :="";
i16gBypassPressureSensorValue.Description :="new signal";
i16gBypassPressureSensorValue.ErrorReaction := eErrorReaction.ERSIG_DFLT;
i16gBypassPressureSensorValue.ReceiverAdress :=1;
i16gBypassPressureSensorValue.ToolScalingDivisor :=1;
i16gBypassPressureSensorValue.ToolScalingMultiplier :=1;
i16gBypassPressureSensorValue.ToolScalingOffset :=0;
i16gBypassPressureSensorValue.ToolUnit :="";


                
END_METHOD
END_FUNCTION_BLOCK

FUNCTION_BLOCK Msg3C1SendToEvision7MessageClass EXTENDS CanReceiveMessageClass
  VAR_INPUT
    u32MinValueEncodeurMast : UInt32CanSignalClass;
    u32MaxValueEncodeurMast : UInt32CanSignalClass;
    Counter : UInt32CanSignalClass;
  END_VAR

            
          

METHOD SetData
  VAR_INPUT
    CanMsgPointer : POINTER TO CanMessageClass;
  END_VAR
                  IF IsValidPointer(canMsgPointer,'SetData') THEN
	SUPER^.SetData(CanMsgPointer);
	//Set the new data
	u32MinValueEncodeurMast.Value := canMsgPointer^.GetUint32(0);
	u32MaxValueEncodeurMast.Value := canMsgPointer^.GetUint32(32);
	//And increase the counter
	Counter.Value := CanMsgPointer^.Counter.Value;
END_IF

                
END_METHOD

PROPERTY u32MinValueEncodeurMastRawValue : UDINT
GET
                    IF u32MinValueEncodeurMast.AppScalingMultiplier = 0 THEN
	_MatchLog^.Error("Get u32MinValueEncodeurMastRawValue", "Division by Zero!");
	RETURN;
End_IF

u32MinValueEncodeurMastRawValue := TO_UDINT((u32MinValueEncodeurMast.Value - u32MinValueEncodeurMast.AppScalingOffset) * u32MinValueEncodeurMast.AppScalingDivisor / u32MinValueEncodeurMast.AppScalingMultiplier);

                  
END_GET
END_PROPERTY

PROPERTY u32MaxValueEncodeurMastRawValue : UDINT
GET
                    IF u32MaxValueEncodeurMast.AppScalingMultiplier = 0 THEN
	_MatchLog^.Error("Get u32MaxValueEncodeurMastRawValue", "Division by Zero!");
	RETURN;
End_IF

u32MaxValueEncodeurMastRawValue := TO_UDINT((u32MaxValueEncodeurMast.Value - u32MaxValueEncodeurMast.AppScalingOffset) * u32MaxValueEncodeurMast.AppScalingDivisor / u32MaxValueEncodeurMast.AppScalingMultiplier);

                  
END_GET
END_PROPERTY

PROPERTY u32MinValueEncodeurMastToolValue : UDINT
GET
                    IF u32MinValueEncodeurMast.ToolScalingDivisor = 0 OR u32MinValueEncodeurMast.AppScalingMultiplier = 0 THEN
	_MatchLog^.Error("Get u32MinValueEncodeurMastToolValue", "Division by Zero!");
	RETURN;
END_IF

u32MinValueEncodeurMastToolValue := TO_UDINT(((u32MinValueEncodeurMast.Value - u32MinValueEncodeurMast.AppScalingOffset) * u32MinValueEncodeurMast.AppScalingDivisor / u32MinValueEncodeurMast.AppScalingMultiplier * u32MinValueEncodeurMast.ToolScalingMultiplier / u32MinValueEncodeurMast.ToolScalingDivisor) + u32MinValueEncodeurMast.ToolScalingOffset);

                  
END_GET
END_PROPERTY

PROPERTY u32MaxValueEncodeurMastToolValue : UDINT
GET
                    IF u32MaxValueEncodeurMast.ToolScalingDivisor = 0 OR u32MaxValueEncodeurMast.AppScalingMultiplier = 0 THEN
	_MatchLog^.Error("Get u32MaxValueEncodeurMastToolValue", "Division by Zero!");
	RETURN;
END_IF

u32MaxValueEncodeurMastToolValue := TO_UDINT(((u32MaxValueEncodeurMast.Value - u32MaxValueEncodeurMast.AppScalingOffset) * u32MaxValueEncodeurMast.AppScalingDivisor / u32MaxValueEncodeurMast.AppScalingMultiplier * u32MaxValueEncodeurMast.ToolScalingMultiplier / u32MaxValueEncodeurMast.ToolScalingDivisor) + u32MaxValueEncodeurMast.ToolScalingOffset);

                  
END_GET
END_PROPERTY

METHOD InitializeCanSignals
                  u32MinValueEncodeurMast.AppScalingDivisor :=1;
u32MinValueEncodeurMast.AppScalingMultiplier :=1;
u32MinValueEncodeurMast.AppScalingOffset :=0;
u32MinValueEncodeurMast.AppUnit :="";
u32MinValueEncodeurMast.CanDefault :=0;
u32MinValueEncodeurMast.CanInit :=0;
u32MinValueEncodeurMast.CanMax :=VBasic.LibConst.U32_MAX;
u32MinValueEncodeurMast.CanMin :=VBasic.LibConst.U32_MIN;
u32MinValueEncodeurMast.CanUnit :="";
u32MinValueEncodeurMast.Description :="new signal";
u32MinValueEncodeurMast.ErrorReaction := eErrorReaction.ERSIG_DFLT;
u32MinValueEncodeurMast.ReceiverAdress :=1;
u32MinValueEncodeurMast.ToolScalingDivisor :=1;
u32MinValueEncodeurMast.ToolScalingMultiplier :=1;
u32MinValueEncodeurMast.ToolScalingOffset :=0;
u32MinValueEncodeurMast.ToolUnit :="";

u32MaxValueEncodeurMast.AppScalingDivisor :=1;
u32MaxValueEncodeurMast.AppScalingMultiplier :=1;
u32MaxValueEncodeurMast.AppScalingOffset :=0;
u32MaxValueEncodeurMast.AppUnit :="";
u32MaxValueEncodeurMast.CanDefault :=0;
u32MaxValueEncodeurMast.CanInit :=0;
u32MaxValueEncodeurMast.CanMax :=VBasic.LibConst.U32_MAX;
u32MaxValueEncodeurMast.CanMin :=VBasic.LibConst.U32_MIN;
u32MaxValueEncodeurMast.CanUnit :="";
u32MaxValueEncodeurMast.Description :="new signal";
u32MaxValueEncodeurMast.ErrorReaction := eErrorReaction.ERSIG_DFLT;
u32MaxValueEncodeurMast.ReceiverAdress :=1;
u32MaxValueEncodeurMast.ToolScalingDivisor :=1;
u32MaxValueEncodeurMast.ToolScalingMultiplier :=1;
u32MaxValueEncodeurMast.ToolScalingOffset :=0;
u32MaxValueEncodeurMast.ToolUnit :="";


                
END_METHOD
END_FUNCTION_BLOCK

FUNCTION_BLOCK Msg4C1SendToEvision7MessageClass EXTENDS CanReceiveMessageClass
  VAR_INPUT
    u32EncodeurMastMeasureRaw : UInt32CanSignalClass;
    u16EncodeurMastMeasureCentimeter : UInt16CanSignalClass;
    Counter : UInt32CanSignalClass;
  END_VAR

            
          

METHOD SetData
  VAR_INPUT
    CanMsgPointer : POINTER TO CanMessageClass;
  END_VAR
                  IF IsValidPointer(canMsgPointer,'SetData') THEN
	SUPER^.SetData(CanMsgPointer);
	//Set the new data
	u32EncodeurMastMeasureRaw.Value := canMsgPointer^.GetUint32(0);
	u16EncodeurMastMeasureCentimeter.Value := canMsgPointer^.GetUint16(32);
	//And increase the counter
	Counter.Value := CanMsgPointer^.Counter.Value;
END_IF

                
END_METHOD

PROPERTY u32EncodeurMastMeasureRawRawValue : UDINT
GET
                    IF u32EncodeurMastMeasureRaw.AppScalingMultiplier = 0 THEN
	_MatchLog^.Error("Get u32EncodeurMastMeasureRawRawValue", "Division by Zero!");
	RETURN;
End_IF

u32EncodeurMastMeasureRawRawValue := TO_UDINT((u32EncodeurMastMeasureRaw.Value - u32EncodeurMastMeasureRaw.AppScalingOffset) * u32EncodeurMastMeasureRaw.AppScalingDivisor / u32EncodeurMastMeasureRaw.AppScalingMultiplier);

                  
END_GET
END_PROPERTY

PROPERTY u16EncodeurMastMeasureCentimeterRawValue : UINT
GET
                    IF u16EncodeurMastMeasureCentimeter.AppScalingMultiplier = 0 THEN
	_MatchLog^.Error("Get u16EncodeurMastMeasureCentimeterRawValue", "Division by Zero!");
	RETURN;
End_IF

u16EncodeurMastMeasureCentimeterRawValue := TO_UINT((u16EncodeurMastMeasureCentimeter.Value - u16EncodeurMastMeasureCentimeter.AppScalingOffset) * u16EncodeurMastMeasureCentimeter.AppScalingDivisor / u16EncodeurMastMeasureCentimeter.AppScalingMultiplier);

                  
END_GET
END_PROPERTY

PROPERTY u32EncodeurMastMeasureRawToolValue : UDINT
GET
                    IF u32EncodeurMastMeasureRaw.ToolScalingDivisor = 0 OR u32EncodeurMastMeasureRaw.AppScalingMultiplier = 0 THEN
	_MatchLog^.Error("Get u32EncodeurMastMeasureRawToolValue", "Division by Zero!");
	RETURN;
END_IF

u32EncodeurMastMeasureRawToolValue := TO_UDINT(((u32EncodeurMastMeasureRaw.Value - u32EncodeurMastMeasureRaw.AppScalingOffset) * u32EncodeurMastMeasureRaw.AppScalingDivisor / u32EncodeurMastMeasureRaw.AppScalingMultiplier * u32EncodeurMastMeasureRaw.ToolScalingMultiplier / u32EncodeurMastMeasureRaw.ToolScalingDivisor) + u32EncodeurMastMeasureRaw.ToolScalingOffset);

                  
END_GET
END_PROPERTY

PROPERTY u16EncodeurMastMeasureCentimeterToolValue : UINT
GET
                    IF u16EncodeurMastMeasureCentimeter.ToolScalingDivisor = 0 OR u16EncodeurMastMeasureCentimeter.AppScalingMultiplier = 0 THEN
	_MatchLog^.Error("Get u16EncodeurMastMeasureCentimeterToolValue", "Division by Zero!");
	RETURN;
END_IF

u16EncodeurMastMeasureCentimeterToolValue := TO_UINT(((u16EncodeurMastMeasureCentimeter.Value - u16EncodeurMastMeasureCentimeter.AppScalingOffset) * u16EncodeurMastMeasureCentimeter.AppScalingDivisor / u16EncodeurMastMeasureCentimeter.AppScalingMultiplier * u16EncodeurMastMeasureCentimeter.ToolScalingMultiplier / u16EncodeurMastMeasureCentimeter.ToolScalingDivisor) + u16EncodeurMastMeasureCentimeter.ToolScalingOffset);

                  
END_GET
END_PROPERTY

METHOD InitializeCanSignals
                  u32EncodeurMastMeasureRaw.AppScalingDivisor :=1;
u32EncodeurMastMeasureRaw.AppScalingMultiplier :=1;
u32EncodeurMastMeasureRaw.AppScalingOffset :=0;
u32EncodeurMastMeasureRaw.AppUnit :="";
u32EncodeurMastMeasureRaw.CanDefault :=0;
u32EncodeurMastMeasureRaw.CanInit :=0;
u32EncodeurMastMeasureRaw.CanMax :=VBasic.LibConst.U32_MAX;
u32EncodeurMastMeasureRaw.CanMin :=VBasic.LibConst.U32_MIN;
u32EncodeurMastMeasureRaw.CanUnit :="";
u32EncodeurMastMeasureRaw.Description :="new signal";
u32EncodeurMastMeasureRaw.ErrorReaction := eErrorReaction.ERSIG_DFLT;
u32EncodeurMastMeasureRaw.ReceiverAdress :=1;
u32EncodeurMastMeasureRaw.ToolScalingDivisor :=1;
u32EncodeurMastMeasureRaw.ToolScalingMultiplier :=1;
u32EncodeurMastMeasureRaw.ToolScalingOffset :=0;
u32EncodeurMastMeasureRaw.ToolUnit :="";

u16EncodeurMastMeasureCentimeter.AppScalingDivisor :=1;
u16EncodeurMastMeasureCentimeter.AppScalingMultiplier :=1;
u16EncodeurMastMeasureCentimeter.AppScalingOffset :=0;
u16EncodeurMastMeasureCentimeter.AppUnit :="";
u16EncodeurMastMeasureCentimeter.CanDefault :=0;
u16EncodeurMastMeasureCentimeter.CanInit :=0;
u16EncodeurMastMeasureCentimeter.CanMax :=VBasic.LibConst.U16_MAX;
u16EncodeurMastMeasureCentimeter.CanMin :=VBasic.LibConst.U16_MIN;
u16EncodeurMastMeasureCentimeter.CanUnit :="";
u16EncodeurMastMeasureCentimeter.Description :="new signal";
u16EncodeurMastMeasureCentimeter.ErrorReaction := eErrorReaction.ERSIG_DFLT;
u16EncodeurMastMeasureCentimeter.ReceiverAdress :=1;
u16EncodeurMastMeasureCentimeter.ToolScalingDivisor :=1;
u16EncodeurMastMeasureCentimeter.ToolScalingMultiplier :=1;
u16EncodeurMastMeasureCentimeter.ToolScalingOffset :=0;
u16EncodeurMastMeasureCentimeter.ToolUnit :="";


                
END_METHOD
END_FUNCTION_BLOCK

FUNCTION_BLOCK Msg5C1SendToEvision7MessageClass EXTENDS CanReceiveMessageClass
  VAR_INPUT
    boReserve0 : BoolCanSignalClass;
    boReserve1 : BoolCanSignalClass;
    boReserve2 : BoolCanSignalClass;
    boReserve3 : BoolCanSignalClass;
    boReserve4 : BoolCanSignalClass;
    boReserve5 : BoolCanSignalClass;
    boReserve6 : BoolCanSignalClass;
    boReserve7 : BoolCanSignalClass;
    boPin107 : BoolCanSignalClass;
    boPin131 : BoolCanSignalClass;
    boPin108 : BoolCanSignalClass;
    boPin132 : BoolCanSignalClass;
    boPin109 : BoolCanSignalClass;
    boPin133 : BoolCanSignalClass;
    boPin110 : BoolCanSignalClass;
    boPin134 : BoolCanSignalClass;
    boPin111 : BoolCanSignalClass;
    boPin135 : BoolCanSignalClass;
    boPin112 : BoolCanSignalClass;
    boPin136 : BoolCanSignalClass;
    boPin113 : BoolCanSignalClass;
    boPin137 : BoolCanSignalClass;
    boPin114 : BoolCanSignalClass;
    boPin138 : BoolCanSignalClass;
    boPin140 : BoolCanSignalClass;
    boPin117 : BoolCanSignalClass;
    boPin141 : BoolCanSignalClass;
    boPin124 : BoolCanSignalClass;
    boPin148 : BoolCanSignalClass;
    boPin153 : BoolCanSignalClass;
    boPin177 : BoolCanSignalClass;
    boPin159 : BoolCanSignalClass;
    boPin183 : BoolCanSignalClass;
    boPin154 : BoolCanSignalClass;
    boPin178 : BoolCanSignalClass;
    boPin157 : BoolCanSignalClass;
    boPin181 : BoolCanSignalClass;
    boPin160 : BoolCanSignalClass;
    boPin184 : BoolCanSignalClass;
    boPin187 : BoolCanSignalClass;
    boPin163 : BoolCanSignalClass;
    boPin149 : BoolCanSignalClass;
    boPin173 : BoolCanSignalClass;
    boPin152 : BoolCanSignalClass;
    boPin176 : BoolCanSignalClass;
    boPin155 : BoolCanSignalClass;
    boPin179 : BoolCanSignalClass;
    boPin158 : BoolCanSignalClass;
    boPin182 : BoolCanSignalClass;
    boPin251 : BoolCanSignalClass;
    boPin186 : BoolCanSignalClass;
    boPin239 : BoolCanSignalClass;
    Counter : UInt32CanSignalClass;
  END_VAR

            
          

METHOD SetData
  VAR_INPUT
    CanMsgPointer : POINTER TO CanMessageClass;
  END_VAR
                  IF IsValidPointer(canMsgPointer,'SetData') THEN
	SUPER^.SetData(CanMsgPointer);
	//Set the new data
	boReserve0.Value := canMsgPointer^.GetBoolOnBit(0);
	boReserve1.Value := canMsgPointer^.GetBoolOnBit(1);
	boReserve2.Value := canMsgPointer^.GetBoolOnBit(2);
	boReserve3.Value := canMsgPointer^.GetBoolOnBit(3);
	boReserve4.Value := canMsgPointer^.GetBoolOnBit(4);
	boReserve5.Value := canMsgPointer^.GetBoolOnBit(5);
	boReserve6.Value := canMsgPointer^.GetBoolOnBit(6);
	boReserve7.Value := canMsgPointer^.GetBoolOnBit(7);
	boPin107.Value := canMsgPointer^.GetBoolOnBit(8);
	boPin131.Value := canMsgPointer^.GetBoolOnBit(9);
	boPin108.Value := canMsgPointer^.GetBoolOnBit(10);
	boPin132.Value := canMsgPointer^.GetBoolOnBit(11);
	boPin109.Value := canMsgPointer^.GetBoolOnBit(12);
	boPin133.Value := canMsgPointer^.GetBoolOnBit(13);
	boPin110.Value := canMsgPointer^.GetBoolOnBit(14);
	boPin134.Value := canMsgPointer^.GetBoolOnBit(15);
	boPin111.Value := canMsgPointer^.GetBoolOnBit(16);
	boPin135.Value := canMsgPointer^.GetBoolOnBit(17);
	boPin112.Value := canMsgPointer^.GetBoolOnBit(18);
	boPin136.Value := canMsgPointer^.GetBoolOnBit(19);
	boPin113.Value := canMsgPointer^.GetBoolOnBit(20);
	boPin137.Value := canMsgPointer^.GetBoolOnBit(21);
	boPin114.Value := canMsgPointer^.GetBoolOnBit(22);
	boPin138.Value := canMsgPointer^.GetBoolOnBit(23);
	boPin140.Value := canMsgPointer^.GetBoolOnBit(24);
	boPin117.Value := canMsgPointer^.GetBoolOnBit(25);
	boPin141.Value := canMsgPointer^.GetBoolOnBit(26);
	boPin124.Value := canMsgPointer^.GetBoolOnBit(27);
	boPin148.Value := canMsgPointer^.GetBoolOnBit(28);
	boPin153.Value := canMsgPointer^.GetBoolOnBit(29);
	boPin177.Value := canMsgPointer^.GetBoolOnBit(30);
	boPin159.Value := canMsgPointer^.GetBoolOnBit(31);
	boPin183.Value := canMsgPointer^.GetBoolOnBit(32);
	boPin154.Value := canMsgPointer^.GetBoolOnBit(33);
	boPin178.Value := canMsgPointer^.GetBoolOnBit(34);
	boPin157.Value := canMsgPointer^.GetBoolOnBit(35);
	boPin181.Value := canMsgPointer^.GetBoolOnBit(36);
	boPin160.Value := canMsgPointer^.GetBoolOnBit(37);
	boPin184.Value := canMsgPointer^.GetBoolOnBit(38);
	boPin187.Value := canMsgPointer^.GetBoolOnBit(39);
	boPin163.Value := canMsgPointer^.GetBoolOnBit(40);
	boPin149.Value := canMsgPointer^.GetBoolOnBit(41);
	boPin173.Value := canMsgPointer^.GetBoolOnBit(42);
	boPin152.Value := canMsgPointer^.GetBoolOnBit(43);
	boPin176.Value := canMsgPointer^.GetBoolOnBit(44);
	boPin155.Value := canMsgPointer^.GetBoolOnBit(45);
	boPin179.Value := canMsgPointer^.GetBoolOnBit(46);
	boPin158.Value := canMsgPointer^.GetBoolOnBit(47);
	boPin182.Value := canMsgPointer^.GetBoolOnBit(48);
	boPin251.Value := canMsgPointer^.GetBoolOnBit(49);
	boPin186.Value := canMsgPointer^.GetBoolOnBit(50);
	boPin239.Value := canMsgPointer^.GetBoolOnBit(51);
	//And increase the counter
	Counter.Value := CanMsgPointer^.Counter.Value;
END_IF

                
END_METHOD

PROPERTY boReserve0RawValue : BOOL
GET
                    boReserve0RawValue := boReserve0.Value;

                  
END_GET
END_PROPERTY

PROPERTY boReserve1RawValue : BOOL
GET
                    boReserve1RawValue := boReserve1.Value;

                  
END_GET
END_PROPERTY

PROPERTY boReserve2RawValue : BOOL
GET
                    boReserve2RawValue := boReserve2.Value;

                  
END_GET
END_PROPERTY

PROPERTY boReserve3RawValue : BOOL
GET
                    boReserve3RawValue := boReserve3.Value;

                  
END_GET
END_PROPERTY

PROPERTY boReserve4RawValue : BOOL
GET
                    boReserve4RawValue := boReserve4.Value;

                  
END_GET
END_PROPERTY

PROPERTY boReserve5RawValue : BOOL
GET
                    boReserve5RawValue := boReserve5.Value;

                  
END_GET
END_PROPERTY

PROPERTY boReserve6RawValue : BOOL
GET
                    boReserve6RawValue := boReserve6.Value;

                  
END_GET
END_PROPERTY

PROPERTY boReserve7RawValue : BOOL
GET
                    boReserve7RawValue := boReserve7.Value;

                  
END_GET
END_PROPERTY

PROPERTY boPin107RawValue : BOOL
GET
                    boPin107RawValue := boPin107.Value;

                  
END_GET
END_PROPERTY

PROPERTY boPin131RawValue : BOOL
GET
                    boPin131RawValue := boPin131.Value;

                  
END_GET
END_PROPERTY

PROPERTY boPin108RawValue : BOOL
GET
                    boPin108RawValue := boPin108.Value;

                  
END_GET
END_PROPERTY

PROPERTY boPin132RawValue : BOOL
GET
                    boPin132RawValue := boPin132.Value;

                  
END_GET
END_PROPERTY

PROPERTY boPin109RawValue : BOOL
GET
                    boPin109RawValue := boPin109.Value;

                  
END_GET
END_PROPERTY

PROPERTY boPin133RawValue : BOOL
GET
                    boPin133RawValue := boPin133.Value;

                  
END_GET
END_PROPERTY

PROPERTY boPin110RawValue : BOOL
GET
                    boPin110RawValue := boPin110.Value;

                  
END_GET
END_PROPERTY

PROPERTY boPin134RawValue : BOOL
GET
                    boPin134RawValue := boPin134.Value;

                  
END_GET
END_PROPERTY

PROPERTY boPin111RawValue : BOOL
GET
                    boPin111RawValue := boPin111.Value;

                  
END_GET
END_PROPERTY

PROPERTY boPin135RawValue : BOOL
GET
                    boPin135RawValue := boPin135.Value;

                  
END_GET
END_PROPERTY

PROPERTY boPin112RawValue : BOOL
GET
                    boPin112RawValue := boPin112.Value;

                  
END_GET
END_PROPERTY

PROPERTY boPin136RawValue : BOOL
GET
                    boPin136RawValue := boPin136.Value;

                  
END_GET
END_PROPERTY

PROPERTY boPin113RawValue : BOOL
GET
                    boPin113RawValue := boPin113.Value;

                  
END_GET
END_PROPERTY

PROPERTY boPin137RawValue : BOOL
GET
                    boPin137RawValue := boPin137.Value;

                  
END_GET
END_PROPERTY

PROPERTY boPin114RawValue : BOOL
GET
                    boPin114RawValue := boPin114.Value;

                  
END_GET
END_PROPERTY

PROPERTY boPin138RawValue : BOOL
GET
                    boPin138RawValue := boPin138.Value;

                  
END_GET
END_PROPERTY

PROPERTY boPin140RawValue : BOOL
GET
                    boPin140RawValue := boPin140.Value;

                  
END_GET
END_PROPERTY

PROPERTY boPin117RawValue : BOOL
GET
                    boPin117RawValue := boPin117.Value;

                  
END_GET
END_PROPERTY

PROPERTY boPin141RawValue : BOOL
GET
                    boPin141RawValue := boPin141.Value;

                  
END_GET
END_PROPERTY

PROPERTY boPin124RawValue : BOOL
GET
                    boPin124RawValue := boPin124.Value;

                  
END_GET
END_PROPERTY

PROPERTY boPin148RawValue : BOOL
GET
                    boPin148RawValue := boPin148.Value;

                  
END_GET
END_PROPERTY

PROPERTY boPin153RawValue : BOOL
GET
                    boPin153RawValue := boPin153.Value;

                  
END_GET
END_PROPERTY

PROPERTY boPin177RawValue : BOOL
GET
                    boPin177RawValue := boPin177.Value;

                  
END_GET
END_PROPERTY

PROPERTY boPin159RawValue : BOOL
GET
                    boPin159RawValue := boPin159.Value;

                  
END_GET
END_PROPERTY

PROPERTY boPin183RawValue : BOOL
GET
                    boPin183RawValue := boPin183.Value;

                  
END_GET
END_PROPERTY

PROPERTY boPin154RawValue : BOOL
GET
                    boPin154RawValue := boPin154.Value;

                  
END_GET
END_PROPERTY

PROPERTY boPin178RawValue : BOOL
GET
                    boPin178RawValue := boPin178.Value;

                  
END_GET
END_PROPERTY

PROPERTY boPin157RawValue : BOOL
GET
                    boPin157RawValue := boPin157.Value;

                  
END_GET
END_PROPERTY

PROPERTY boPin181RawValue : BOOL
GET
                    boPin181RawValue := boPin181.Value;

                  
END_GET
END_PROPERTY

PROPERTY boPin160RawValue : BOOL
GET
                    boPin160RawValue := boPin160.Value;

                  
END_GET
END_PROPERTY

PROPERTY boPin184RawValue : BOOL
GET
                    boPin184RawValue := boPin184.Value;

                  
END_GET
END_PROPERTY

PROPERTY boPin187RawValue : BOOL
GET
                    boPin187RawValue := boPin187.Value;

                  
END_GET
END_PROPERTY

PROPERTY boPin163RawValue : BOOL
GET
                    boPin163RawValue := boPin163.Value;

                  
END_GET
END_PROPERTY

PROPERTY boPin149RawValue : BOOL
GET
                    boPin149RawValue := boPin149.Value;

                  
END_GET
END_PROPERTY

PROPERTY boPin173RawValue : BOOL
GET
                    boPin173RawValue := boPin173.Value;

                  
END_GET
END_PROPERTY

PROPERTY boPin152RawValue : BOOL
GET
                    boPin152RawValue := boPin152.Value;

                  
END_GET
END_PROPERTY

PROPERTY boPin176RawValue : BOOL
GET
                    boPin176RawValue := boPin176.Value;

                  
END_GET
END_PROPERTY

PROPERTY boPin155RawValue : BOOL
GET
                    boPin155RawValue := boPin155.Value;

                  
END_GET
END_PROPERTY

PROPERTY boPin179RawValue : BOOL
GET
                    boPin179RawValue := boPin179.Value;

                  
END_GET
END_PROPERTY

PROPERTY boPin158RawValue : BOOL
GET
                    boPin158RawValue := boPin158.Value;

                  
END_GET
END_PROPERTY

PROPERTY boPin182RawValue : BOOL
GET
                    boPin182RawValue := boPin182.Value;

                  
END_GET
END_PROPERTY

PROPERTY boPin251RawValue : BOOL
GET
                    boPin251RawValue := boPin251.Value;

                  
END_GET
END_PROPERTY

PROPERTY boPin186RawValue : BOOL
GET
                    boPin186RawValue := boPin186.Value;

                  
END_GET
END_PROPERTY

PROPERTY boPin239RawValue : BOOL
GET
                    boPin239RawValue := boPin239.Value;

                  
END_GET
END_PROPERTY

PROPERTY boReserve0ToolValue : BOOL
GET
                    boReserve0ToolValue := boReserve0.Value;

                  
END_GET
END_PROPERTY

PROPERTY boReserve1ToolValue : BOOL
GET
                    boReserve1ToolValue := boReserve1.Value;

                  
END_GET
END_PROPERTY

PROPERTY boReserve2ToolValue : BOOL
GET
                    boReserve2ToolValue := boReserve2.Value;

                  
END_GET
END_PROPERTY

PROPERTY boReserve3ToolValue : BOOL
GET
                    boReserve3ToolValue := boReserve3.Value;

                  
END_GET
END_PROPERTY

PROPERTY boReserve4ToolValue : BOOL
GET
                    boReserve4ToolValue := boReserve4.Value;

                  
END_GET
END_PROPERTY

PROPERTY boReserve5ToolValue : BOOL
GET
                    boReserve5ToolValue := boReserve5.Value;

                  
END_GET
END_PROPERTY

PROPERTY boReserve6ToolValue : BOOL
GET
                    boReserve6ToolValue := boReserve6.Value;

                  
END_GET
END_PROPERTY

PROPERTY boReserve7ToolValue : BOOL
GET
                    boReserve7ToolValue := boReserve7.Value;

                  
END_GET
END_PROPERTY

PROPERTY boPin107ToolValue : BOOL
GET
                    boPin107ToolValue := boPin107.Value;

                  
END_GET
END_PROPERTY

PROPERTY boPin131ToolValue : BOOL
GET
                    boPin131ToolValue := boPin131.Value;

                  
END_GET
END_PROPERTY

PROPERTY boPin108ToolValue : BOOL
GET
                    boPin108ToolValue := boPin108.Value;

                  
END_GET
END_PROPERTY

PROPERTY boPin132ToolValue : BOOL
GET
                    boPin132ToolValue := boPin132.Value;

                  
END_GET
END_PROPERTY

PROPERTY boPin109ToolValue : BOOL
GET
                    boPin109ToolValue := boPin109.Value;

                  
END_GET
END_PROPERTY

PROPERTY boPin133ToolValue : BOOL
GET
                    boPin133ToolValue := boPin133.Value;

                  
END_GET
END_PROPERTY

PROPERTY boPin110ToolValue : BOOL
GET
                    boPin110ToolValue := boPin110.Value;

                  
END_GET
END_PROPERTY

PROPERTY boPin134ToolValue : BOOL
GET
                    boPin134ToolValue := boPin134.Value;

                  
END_GET
END_PROPERTY

PROPERTY boPin111ToolValue : BOOL
GET
                    boPin111ToolValue := boPin111.Value;

                  
END_GET
END_PROPERTY

PROPERTY boPin135ToolValue : BOOL
GET
                    boPin135ToolValue := boPin135.Value;

                  
END_GET
END_PROPERTY

PROPERTY boPin112ToolValue : BOOL
GET
                    boPin112ToolValue := boPin112.Value;

                  
END_GET
END_PROPERTY

PROPERTY boPin136ToolValue : BOOL
GET
                    boPin136ToolValue := boPin136.Value;

                  
END_GET
END_PROPERTY

PROPERTY boPin113ToolValue : BOOL
GET
                    boPin113ToolValue := boPin113.Value;

                  
END_GET
END_PROPERTY

PROPERTY boPin137ToolValue : BOOL
GET
                    boPin137ToolValue := boPin137.Value;

                  
END_GET
END_PROPERTY

PROPERTY boPin114ToolValue : BOOL
GET
                    boPin114ToolValue := boPin114.Value;

                  
END_GET
END_PROPERTY

PROPERTY boPin138ToolValue : BOOL
GET
                    boPin138ToolValue := boPin138.Value;

                  
END_GET
END_PROPERTY

PROPERTY boPin140ToolValue : BOOL
GET
                    boPin140ToolValue := boPin140.Value;

                  
END_GET
END_PROPERTY

PROPERTY boPin117ToolValue : BOOL
GET
                    boPin117ToolValue := boPin117.Value;

                  
END_GET
END_PROPERTY

PROPERTY boPin141ToolValue : BOOL
GET
                    boPin141ToolValue := boPin141.Value;

                  
END_GET
END_PROPERTY

PROPERTY boPin124ToolValue : BOOL
GET
                    boPin124ToolValue := boPin124.Value;

                  
END_GET
END_PROPERTY

PROPERTY boPin148ToolValue : BOOL
GET
                    boPin148ToolValue := boPin148.Value;

                  
END_GET
END_PROPERTY

PROPERTY boPin153ToolValue : BOOL
GET
                    boPin153ToolValue := boPin153.Value;

                  
END_GET
END_PROPERTY

PROPERTY boPin177ToolValue : BOOL
GET
                    boPin177ToolValue := boPin177.Value;

                  
END_GET
END_PROPERTY

PROPERTY boPin159ToolValue : BOOL
GET
                    boPin159ToolValue := boPin159.Value;

                  
END_GET
END_PROPERTY

PROPERTY boPin183ToolValue : BOOL
GET
                    boPin183ToolValue := boPin183.Value;

                  
END_GET
END_PROPERTY

PROPERTY boPin154ToolValue : BOOL
GET
                    boPin154ToolValue := boPin154.Value;

                  
END_GET
END_PROPERTY

PROPERTY boPin178ToolValue : BOOL
GET
                    boPin178ToolValue := boPin178.Value;

                  
END_GET
END_PROPERTY

PROPERTY boPin157ToolValue : BOOL
GET
                    boPin157ToolValue := boPin157.Value;

                  
END_GET
END_PROPERTY

PROPERTY boPin181ToolValue : BOOL
GET
                    boPin181ToolValue := boPin181.Value;

                  
END_GET
END_PROPERTY

PROPERTY boPin160ToolValue : BOOL
GET
                    boPin160ToolValue := boPin160.Value;

                  
END_GET
END_PROPERTY

PROPERTY boPin184ToolValue : BOOL
GET
                    boPin184ToolValue := boPin184.Value;

                  
END_GET
END_PROPERTY

PROPERTY boPin187ToolValue : BOOL
GET
                    boPin187ToolValue := boPin187.Value;

                  
END_GET
END_PROPERTY

PROPERTY boPin163ToolValue : BOOL
GET
                    boPin163ToolValue := boPin163.Value;

                  
END_GET
END_PROPERTY

PROPERTY boPin149ToolValue : BOOL
GET
                    boPin149ToolValue := boPin149.Value;

                  
END_GET
END_PROPERTY

PROPERTY boPin173ToolValue : BOOL
GET
                    boPin173ToolValue := boPin173.Value;

                  
END_GET
END_PROPERTY

PROPERTY boPin152ToolValue : BOOL
GET
                    boPin152ToolValue := boPin152.Value;

                  
END_GET
END_PROPERTY

PROPERTY boPin176ToolValue : BOOL
GET
                    boPin176ToolValue := boPin176.Value;

                  
END_GET
END_PROPERTY

PROPERTY boPin155ToolValue : BOOL
GET
                    boPin155ToolValue := boPin155.Value;

                  
END_GET
END_PROPERTY

PROPERTY boPin179ToolValue : BOOL
GET
                    boPin179ToolValue := boPin179.Value;

                  
END_GET
END_PROPERTY

PROPERTY boPin158ToolValue : BOOL
GET
                    boPin158ToolValue := boPin158.Value;

                  
END_GET
END_PROPERTY

PROPERTY boPin182ToolValue : BOOL
GET
                    boPin182ToolValue := boPin182.Value;

                  
END_GET
END_PROPERTY

PROPERTY boPin251ToolValue : BOOL
GET
                    boPin251ToolValue := boPin251.Value;

                  
END_GET
END_PROPERTY

PROPERTY boPin186ToolValue : BOOL
GET
                    boPin186ToolValue := boPin186.Value;

                  
END_GET
END_PROPERTY

PROPERTY boPin239ToolValue : BOOL
GET
                    boPin239ToolValue := boPin239.Value;

                  
END_GET
END_PROPERTY

METHOD InitializeCanSignals
                  boReserve0.AppScalingDivisor :=1;
boReserve0.AppScalingMultiplier :=1;
boReserve0.AppScalingOffset :=0;
boReserve0.AppUnit :="";
boReserve0.CanDefault :=0;
boReserve0.CanInit :=0;
boReserve0.CanMax :=1;
boReserve0.CanMin :=0;
boReserve0.CanUnit :="";
boReserve0.Description :="for the Neotec diag pages";
boReserve0.ErrorReaction := eErrorReaction.ERSIG_DFLT;
boReserve0.ReceiverAdress :=1;
boReserve0.ToolScalingDivisor :=1;
boReserve0.ToolScalingMultiplier :=1;
boReserve0.ToolScalingOffset :=0;
boReserve0.ToolUnit :="";

boReserve1.AppScalingDivisor :=1;
boReserve1.AppScalingMultiplier :=1;
boReserve1.AppScalingOffset :=0;
boReserve1.AppUnit :="";
boReserve1.CanDefault :=0;
boReserve1.CanInit :=0;
boReserve1.CanMax :=1;
boReserve1.CanMin :=0;
boReserve1.CanUnit :="";
boReserve1.Description :="for the Neotec diag pages";
boReserve1.ErrorReaction := eErrorReaction.ERSIG_DFLT;
boReserve1.ReceiverAdress :=1;
boReserve1.ToolScalingDivisor :=1;
boReserve1.ToolScalingMultiplier :=1;
boReserve1.ToolScalingOffset :=0;
boReserve1.ToolUnit :="";

boReserve2.AppScalingDivisor :=1;
boReserve2.AppScalingMultiplier :=1;
boReserve2.AppScalingOffset :=0;
boReserve2.AppUnit :="";
boReserve2.CanDefault :=0;
boReserve2.CanInit :=0;
boReserve2.CanMax :=1;
boReserve2.CanMin :=0;
boReserve2.CanUnit :="";
boReserve2.Description :="for the Neotec diag pages";
boReserve2.ErrorReaction := eErrorReaction.ERSIG_DFLT;
boReserve2.ReceiverAdress :=1;
boReserve2.ToolScalingDivisor :=1;
boReserve2.ToolScalingMultiplier :=1;
boReserve2.ToolScalingOffset :=0;
boReserve2.ToolUnit :="";

boReserve3.AppScalingDivisor :=1;
boReserve3.AppScalingMultiplier :=1;
boReserve3.AppScalingOffset :=0;
boReserve3.AppUnit :="";
boReserve3.CanDefault :=0;
boReserve3.CanInit :=0;
boReserve3.CanMax :=1;
boReserve3.CanMin :=0;
boReserve3.CanUnit :="";
boReserve3.Description :="for the Neotec diag pages";
boReserve3.ErrorReaction := eErrorReaction.ERSIG_DFLT;
boReserve3.ReceiverAdress :=1;
boReserve3.ToolScalingDivisor :=1;
boReserve3.ToolScalingMultiplier :=1;
boReserve3.ToolScalingOffset :=0;
boReserve3.ToolUnit :="";

boReserve4.AppScalingDivisor :=1;
boReserve4.AppScalingMultiplier :=1;
boReserve4.AppScalingOffset :=0;
boReserve4.AppUnit :="";
boReserve4.CanDefault :=0;
boReserve4.CanInit :=0;
boReserve4.CanMax :=1;
boReserve4.CanMin :=0;
boReserve4.CanUnit :="";
boReserve4.Description :="for the Neotec diag pages";
boReserve4.ErrorReaction := eErrorReaction.ERSIG_DFLT;
boReserve4.ReceiverAdress :=1;
boReserve4.ToolScalingDivisor :=1;
boReserve4.ToolScalingMultiplier :=1;
boReserve4.ToolScalingOffset :=0;
boReserve4.ToolUnit :="";

boReserve5.AppScalingDivisor :=1;
boReserve5.AppScalingMultiplier :=1;
boReserve5.AppScalingOffset :=0;
boReserve5.AppUnit :="";
boReserve5.CanDefault :=0;
boReserve5.CanInit :=0;
boReserve5.CanMax :=1;
boReserve5.CanMin :=0;
boReserve5.CanUnit :="";
boReserve5.Description :="for the Neotec diag pages";
boReserve5.ErrorReaction := eErrorReaction.ERSIG_DFLT;
boReserve5.ReceiverAdress :=1;
boReserve5.ToolScalingDivisor :=1;
boReserve5.ToolScalingMultiplier :=1;
boReserve5.ToolScalingOffset :=0;
boReserve5.ToolUnit :="";

boReserve6.AppScalingDivisor :=1;
boReserve6.AppScalingMultiplier :=1;
boReserve6.AppScalingOffset :=0;
boReserve6.AppUnit :="";
boReserve6.CanDefault :=0;
boReserve6.CanInit :=0;
boReserve6.CanMax :=1;
boReserve6.CanMin :=0;
boReserve6.CanUnit :="";
boReserve6.Description :="for the Neotec diag pages";
boReserve6.ErrorReaction := eErrorReaction.ERSIG_DFLT;
boReserve6.ReceiverAdress :=1;
boReserve6.ToolScalingDivisor :=1;
boReserve6.ToolScalingMultiplier :=1;
boReserve6.ToolScalingOffset :=0;
boReserve6.ToolUnit :="";

boReserve7.AppScalingDivisor :=1;
boReserve7.AppScalingMultiplier :=1;
boReserve7.AppScalingOffset :=0;
boReserve7.AppUnit :="";
boReserve7.CanDefault :=0;
boReserve7.CanInit :=0;
boReserve7.CanMax :=1;
boReserve7.CanMin :=0;
boReserve7.CanUnit :="";
boReserve7.Description :="for the Neotec diag pages";
boReserve7.ErrorReaction := eErrorReaction.ERSIG_DFLT;
boReserve7.ReceiverAdress :=1;
boReserve7.ToolScalingDivisor :=1;
boReserve7.ToolScalingMultiplier :=1;
boReserve7.ToolScalingOffset :=0;
boReserve7.ToolUnit :="";

boPin107.AppScalingDivisor :=1;
boPin107.AppScalingMultiplier :=1;
boPin107.AppScalingOffset :=0;
boPin107.AppUnit :="";
boPin107.CanDefault :=0;
boPin107.CanInit :=0;
boPin107.CanMax :=1;
boPin107.CanMin :=0;
boPin107.CanUnit :="";
boPin107.Description :="for the Neotec diag pages";
boPin107.ErrorReaction := eErrorReaction.ERSIG_DFLT;
boPin107.ReceiverAdress :=1;
boPin107.ToolScalingDivisor :=1;
boPin107.ToolScalingMultiplier :=1;
boPin107.ToolScalingOffset :=0;
boPin107.ToolUnit :="";

boPin131.AppScalingDivisor :=1;
boPin131.AppScalingMultiplier :=1;
boPin131.AppScalingOffset :=0;
boPin131.AppUnit :="";
boPin131.CanDefault :=0;
boPin131.CanInit :=0;
boPin131.CanMax :=1;
boPin131.CanMin :=0;
boPin131.CanUnit :="";
boPin131.Description :="for the Neotec diag pages";
boPin131.ErrorReaction := eErrorReaction.ERSIG_DFLT;
boPin131.ReceiverAdress :=1;
boPin131.ToolScalingDivisor :=1;
boPin131.ToolScalingMultiplier :=1;
boPin131.ToolScalingOffset :=0;
boPin131.ToolUnit :="";

boPin108.AppScalingDivisor :=1;
boPin108.AppScalingMultiplier :=1;
boPin108.AppScalingOffset :=0;
boPin108.AppUnit :="";
boPin108.CanDefault :=0;
boPin108.CanInit :=0;
boPin108.CanMax :=1;
boPin108.CanMin :=0;
boPin108.CanUnit :="";
boPin108.Description :="for the Neotec diag pages";
boPin108.ErrorReaction := eErrorReaction.ERSIG_DFLT;
boPin108.ReceiverAdress :=1;
boPin108.ToolScalingDivisor :=1;
boPin108.ToolScalingMultiplier :=1;
boPin108.ToolScalingOffset :=0;
boPin108.ToolUnit :="";

boPin132.AppScalingDivisor :=1;
boPin132.AppScalingMultiplier :=1;
boPin132.AppScalingOffset :=0;
boPin132.AppUnit :="";
boPin132.CanDefault :=0;
boPin132.CanInit :=0;
boPin132.CanMax :=1;
boPin132.CanMin :=0;
boPin132.CanUnit :="";
boPin132.Description :="for the Neotec diag pages";
boPin132.ErrorReaction := eErrorReaction.ERSIG_DFLT;
boPin132.ReceiverAdress :=1;
boPin132.ToolScalingDivisor :=1;
boPin132.ToolScalingMultiplier :=1;
boPin132.ToolScalingOffset :=0;
boPin132.ToolUnit :="";

boPin109.AppScalingDivisor :=1;
boPin109.AppScalingMultiplier :=1;
boPin109.AppScalingOffset :=0;
boPin109.AppUnit :="";
boPin109.CanDefault :=0;
boPin109.CanInit :=0;
boPin109.CanMax :=1;
boPin109.CanMin :=0;
boPin109.CanUnit :="";
boPin109.Description :="for the Neotec diag pages";
boPin109.ErrorReaction := eErrorReaction.ERSIG_DFLT;
boPin109.ReceiverAdress :=1;
boPin109.ToolScalingDivisor :=1;
boPin109.ToolScalingMultiplier :=1;
boPin109.ToolScalingOffset :=0;
boPin109.ToolUnit :="";

boPin133.AppScalingDivisor :=1;
boPin133.AppScalingMultiplier :=1;
boPin133.AppScalingOffset :=0;
boPin133.AppUnit :="";
boPin133.CanDefault :=0;
boPin133.CanInit :=0;
boPin133.CanMax :=1;
boPin133.CanMin :=0;
boPin133.CanUnit :="";
boPin133.Description :="for the Neotec diag pages";
boPin133.ErrorReaction := eErrorReaction.ERSIG_DFLT;
boPin133.ReceiverAdress :=1;
boPin133.ToolScalingDivisor :=1;
boPin133.ToolScalingMultiplier :=1;
boPin133.ToolScalingOffset :=0;
boPin133.ToolUnit :="";

boPin110.AppScalingDivisor :=1;
boPin110.AppScalingMultiplier :=1;
boPin110.AppScalingOffset :=0;
boPin110.AppUnit :="";
boPin110.CanDefault :=0;
boPin110.CanInit :=0;
boPin110.CanMax :=1;
boPin110.CanMin :=0;
boPin110.CanUnit :="";
boPin110.Description :="for the Neotec diag pages";
boPin110.ErrorReaction := eErrorReaction.ERSIG_DFLT;
boPin110.ReceiverAdress :=1;
boPin110.ToolScalingDivisor :=1;
boPin110.ToolScalingMultiplier :=1;
boPin110.ToolScalingOffset :=0;
boPin110.ToolUnit :="";

boPin134.AppScalingDivisor :=1;
boPin134.AppScalingMultiplier :=1;
boPin134.AppScalingOffset :=0;
boPin134.AppUnit :="";
boPin134.CanDefault :=0;
boPin134.CanInit :=0;
boPin134.CanMax :=1;
boPin134.CanMin :=0;
boPin134.CanUnit :="";
boPin134.Description :="for the Neotec diag pages";
boPin134.ErrorReaction := eErrorReaction.ERSIG_DFLT;
boPin134.ReceiverAdress :=1;
boPin134.ToolScalingDivisor :=1;
boPin134.ToolScalingMultiplier :=1;
boPin134.ToolScalingOffset :=0;
boPin134.ToolUnit :="";

boPin111.AppScalingDivisor :=1;
boPin111.AppScalingMultiplier :=1;
boPin111.AppScalingOffset :=0;
boPin111.AppUnit :="";
boPin111.CanDefault :=0;
boPin111.CanInit :=0;
boPin111.CanMax :=1;
boPin111.CanMin :=0;
boPin111.CanUnit :="";
boPin111.Description :="for the Neotec diag pages";
boPin111.ErrorReaction := eErrorReaction.ERSIG_DFLT;
boPin111.ReceiverAdress :=1;
boPin111.ToolScalingDivisor :=1;
boPin111.ToolScalingMultiplier :=1;
boPin111.ToolScalingOffset :=0;
boPin111.ToolUnit :="";

boPin135.AppScalingDivisor :=1;
boPin135.AppScalingMultiplier :=1;
boPin135.AppScalingOffset :=0;
boPin135.AppUnit :="";
boPin135.CanDefault :=0;
boPin135.CanInit :=0;
boPin135.CanMax :=1;
boPin135.CanMin :=0;
boPin135.CanUnit :="";
boPin135.Description :="for the Neotec diag pages";
boPin135.ErrorReaction := eErrorReaction.ERSIG_DFLT;
boPin135.ReceiverAdress :=1;
boPin135.ToolScalingDivisor :=1;
boPin135.ToolScalingMultiplier :=1;
boPin135.ToolScalingOffset :=0;
boPin135.ToolUnit :="";

boPin112.AppScalingDivisor :=1;
boPin112.AppScalingMultiplier :=1;
boPin112.AppScalingOffset :=0;
boPin112.AppUnit :="";
boPin112.CanDefault :=0;
boPin112.CanInit :=0;
boPin112.CanMax :=1;
boPin112.CanMin :=0;
boPin112.CanUnit :="";
boPin112.Description :="for the Neotec diag pages";
boPin112.ErrorReaction := eErrorReaction.ERSIG_DFLT;
boPin112.ReceiverAdress :=1;
boPin112.ToolScalingDivisor :=1;
boPin112.ToolScalingMultiplier :=1;
boPin112.ToolScalingOffset :=0;
boPin112.ToolUnit :="";

boPin136.AppScalingDivisor :=1;
boPin136.AppScalingMultiplier :=1;
boPin136.AppScalingOffset :=0;
boPin136.AppUnit :="";
boPin136.CanDefault :=0;
boPin136.CanInit :=0;
boPin136.CanMax :=1;
boPin136.CanMin :=0;
boPin136.CanUnit :="";
boPin136.Description :="for the Neotec diag pages";
boPin136.ErrorReaction := eErrorReaction.ERSIG_DFLT;
boPin136.ReceiverAdress :=1;
boPin136.ToolScalingDivisor :=1;
boPin136.ToolScalingMultiplier :=1;
boPin136.ToolScalingOffset :=0;
boPin136.ToolUnit :="";

boPin113.AppScalingDivisor :=1;
boPin113.AppScalingMultiplier :=1;
boPin113.AppScalingOffset :=0;
boPin113.AppUnit :="";
boPin113.CanDefault :=0;
boPin113.CanInit :=0;
boPin113.CanMax :=1;
boPin113.CanMin :=0;
boPin113.CanUnit :="";
boPin113.Description :="for the Neotec diag pages";
boPin113.ErrorReaction := eErrorReaction.ERSIG_DFLT;
boPin113.ReceiverAdress :=1;
boPin113.ToolScalingDivisor :=1;
boPin113.ToolScalingMultiplier :=1;
boPin113.ToolScalingOffset :=0;
boPin113.ToolUnit :="";

boPin137.AppScalingDivisor :=1;
boPin137.AppScalingMultiplier :=1;
boPin137.AppScalingOffset :=0;
boPin137.AppUnit :="";
boPin137.CanDefault :=0;
boPin137.CanInit :=0;
boPin137.CanMax :=1;
boPin137.CanMin :=0;
boPin137.CanUnit :="";
boPin137.Description :="for the Neotec diag pages";
boPin137.ErrorReaction := eErrorReaction.ERSIG_DFLT;
boPin137.ReceiverAdress :=1;
boPin137.ToolScalingDivisor :=1;
boPin137.ToolScalingMultiplier :=1;
boPin137.ToolScalingOffset :=0;
boPin137.ToolUnit :="";

boPin114.AppScalingDivisor :=1;
boPin114.AppScalingMultiplier :=1;
boPin114.AppScalingOffset :=0;
boPin114.AppUnit :="";
boPin114.CanDefault :=0;
boPin114.CanInit :=0;
boPin114.CanMax :=1;
boPin114.CanMin :=0;
boPin114.CanUnit :="";
boPin114.Description :="for the Neotec diag pages";
boPin114.ErrorReaction := eErrorReaction.ERSIG_DFLT;
boPin114.ReceiverAdress :=1;
boPin114.ToolScalingDivisor :=1;
boPin114.ToolScalingMultiplier :=1;
boPin114.ToolScalingOffset :=0;
boPin114.ToolUnit :="";

boPin138.AppScalingDivisor :=1;
boPin138.AppScalingMultiplier :=1;
boPin138.AppScalingOffset :=0;
boPin138.AppUnit :="";
boPin138.CanDefault :=0;
boPin138.CanInit :=0;
boPin138.CanMax :=1;
boPin138.CanMin :=0;
boPin138.CanUnit :="";
boPin138.Description :="for the Neotec diag pages";
boPin138.ErrorReaction := eErrorReaction.ERSIG_DFLT;
boPin138.ReceiverAdress :=1;
boPin138.ToolScalingDivisor :=1;
boPin138.ToolScalingMultiplier :=1;
boPin138.ToolScalingOffset :=0;
boPin138.ToolUnit :="";

boPin140.AppScalingDivisor :=1;
boPin140.AppScalingMultiplier :=1;
boPin140.AppScalingOffset :=0;
boPin140.AppUnit :="";
boPin140.CanDefault :=0;
boPin140.CanInit :=0;
boPin140.CanMax :=1;
boPin140.CanMin :=0;
boPin140.CanUnit :="";
boPin140.Description :="for the Neotec diag pages";
boPin140.ErrorReaction := eErrorReaction.ERSIG_DFLT;
boPin140.ReceiverAdress :=1;
boPin140.ToolScalingDivisor :=1;
boPin140.ToolScalingMultiplier :=1;
boPin140.ToolScalingOffset :=0;
boPin140.ToolUnit :="";

boPin117.AppScalingDivisor :=1;
boPin117.AppScalingMultiplier :=1;
boPin117.AppScalingOffset :=0;
boPin117.AppUnit :="";
boPin117.CanDefault :=0;
boPin117.CanInit :=0;
boPin117.CanMax :=1;
boPin117.CanMin :=0;
boPin117.CanUnit :="";
boPin117.Description :="for the Neotec diag pages";
boPin117.ErrorReaction := eErrorReaction.ERSIG_DFLT;
boPin117.ReceiverAdress :=1;
boPin117.ToolScalingDivisor :=1;
boPin117.ToolScalingMultiplier :=1;
boPin117.ToolScalingOffset :=0;
boPin117.ToolUnit :="";

boPin141.AppScalingDivisor :=1;
boPin141.AppScalingMultiplier :=1;
boPin141.AppScalingOffset :=0;
boPin141.AppUnit :="";
boPin141.CanDefault :=0;
boPin141.CanInit :=0;
boPin141.CanMax :=1;
boPin141.CanMin :=0;
boPin141.CanUnit :="";
boPin141.Description :="for the Neotec diag pages";
boPin141.ErrorReaction := eErrorReaction.ERSIG_DFLT;
boPin141.ReceiverAdress :=1;
boPin141.ToolScalingDivisor :=1;
boPin141.ToolScalingMultiplier :=1;
boPin141.ToolScalingOffset :=0;
boPin141.ToolUnit :="";

boPin124.AppScalingDivisor :=1;
boPin124.AppScalingMultiplier :=1;
boPin124.AppScalingOffset :=0;
boPin124.AppUnit :="";
boPin124.CanDefault :=0;
boPin124.CanInit :=0;
boPin124.CanMax :=1;
boPin124.CanMin :=0;
boPin124.CanUnit :="";
boPin124.Description :="for the Neotec diag pages";
boPin124.ErrorReaction := eErrorReaction.ERSIG_DFLT;
boPin124.ReceiverAdress :=1;
boPin124.ToolScalingDivisor :=1;
boPin124.ToolScalingMultiplier :=1;
boPin124.ToolScalingOffset :=0;
boPin124.ToolUnit :="";

boPin148.AppScalingDivisor :=1;
boPin148.AppScalingMultiplier :=1;
boPin148.AppScalingOffset :=0;
boPin148.AppUnit :="";
boPin148.CanDefault :=0;
boPin148.CanInit :=0;
boPin148.CanMax :=1;
boPin148.CanMin :=0;
boPin148.CanUnit :="";
boPin148.Description :="for the Neotec diag pages";
boPin148.ErrorReaction := eErrorReaction.ERSIG_DFLT;
boPin148.ReceiverAdress :=1;
boPin148.ToolScalingDivisor :=1;
boPin148.ToolScalingMultiplier :=1;
boPin148.ToolScalingOffset :=0;
boPin148.ToolUnit :="";

boPin153.AppScalingDivisor :=1;
boPin153.AppScalingMultiplier :=1;
boPin153.AppScalingOffset :=0;
boPin153.AppUnit :="";
boPin153.CanDefault :=0;
boPin153.CanInit :=0;
boPin153.CanMax :=1;
boPin153.CanMin :=0;
boPin153.CanUnit :="";
boPin153.Description :="for the Neotec diag pages";
boPin153.ErrorReaction := eErrorReaction.ERSIG_DFLT;
boPin153.ReceiverAdress :=1;
boPin153.ToolScalingDivisor :=1;
boPin153.ToolScalingMultiplier :=1;
boPin153.ToolScalingOffset :=0;
boPin153.ToolUnit :="";

boPin177.AppScalingDivisor :=1;
boPin177.AppScalingMultiplier :=1;
boPin177.AppScalingOffset :=0;
boPin177.AppUnit :="";
boPin177.CanDefault :=0;
boPin177.CanInit :=0;
boPin177.CanMax :=1;
boPin177.CanMin :=0;
boPin177.CanUnit :="";
boPin177.Description :="for the Neotec diag pages";
boPin177.ErrorReaction := eErrorReaction.ERSIG_DFLT;
boPin177.ReceiverAdress :=1;
boPin177.ToolScalingDivisor :=1;
boPin177.ToolScalingMultiplier :=1;
boPin177.ToolScalingOffset :=0;
boPin177.ToolUnit :="";

boPin159.AppScalingDivisor :=1;
boPin159.AppScalingMultiplier :=1;
boPin159.AppScalingOffset :=0;
boPin159.AppUnit :="";
boPin159.CanDefault :=0;
boPin159.CanInit :=0;
boPin159.CanMax :=1;
boPin159.CanMin :=0;
boPin159.CanUnit :="";
boPin159.Description :="for the Neotec diag pages";
boPin159.ErrorReaction := eErrorReaction.ERSIG_DFLT;
boPin159.ReceiverAdress :=1;
boPin159.ToolScalingDivisor :=1;
boPin159.ToolScalingMultiplier :=1;
boPin159.ToolScalingOffset :=0;
boPin159.ToolUnit :="";

boPin183.AppScalingDivisor :=1;
boPin183.AppScalingMultiplier :=1;
boPin183.AppScalingOffset :=0;
boPin183.AppUnit :="";
boPin183.CanDefault :=0;
boPin183.CanInit :=0;
boPin183.CanMax :=1;
boPin183.CanMin :=0;
boPin183.CanUnit :="";
boPin183.Description :="for the Neotec diag pages";
boPin183.ErrorReaction := eErrorReaction.ERSIG_DFLT;
boPin183.ReceiverAdress :=1;
boPin183.ToolScalingDivisor :=1;
boPin183.ToolScalingMultiplier :=1;
boPin183.ToolScalingOffset :=0;
boPin183.ToolUnit :="";

boPin154.AppScalingDivisor :=1;
boPin154.AppScalingMultiplier :=1;
boPin154.AppScalingOffset :=0;
boPin154.AppUnit :="";
boPin154.CanDefault :=0;
boPin154.CanInit :=0;
boPin154.CanMax :=1;
boPin154.CanMin :=0;
boPin154.CanUnit :="";
boPin154.Description :="for the Neotec diag pages";
boPin154.ErrorReaction := eErrorReaction.ERSIG_DFLT;
boPin154.ReceiverAdress :=1;
boPin154.ToolScalingDivisor :=1;
boPin154.ToolScalingMultiplier :=1;
boPin154.ToolScalingOffset :=0;
boPin154.ToolUnit :="";

boPin178.AppScalingDivisor :=1;
boPin178.AppScalingMultiplier :=1;
boPin178.AppScalingOffset :=0;
boPin178.AppUnit :="";
boPin178.CanDefault :=0;
boPin178.CanInit :=0;
boPin178.CanMax :=1;
boPin178.CanMin :=0;
boPin178.CanUnit :="";
boPin178.Description :="for the Neotec diag pages";
boPin178.ErrorReaction := eErrorReaction.ERSIG_DFLT;
boPin178.ReceiverAdress :=1;
boPin178.ToolScalingDivisor :=1;
boPin178.ToolScalingMultiplier :=1;
boPin178.ToolScalingOffset :=0;
boPin178.ToolUnit :="";

boPin157.AppScalingDivisor :=1;
boPin157.AppScalingMultiplier :=1;
boPin157.AppScalingOffset :=0;
boPin157.AppUnit :="";
boPin157.CanDefault :=0;
boPin157.CanInit :=0;
boPin157.CanMax :=1;
boPin157.CanMin :=0;
boPin157.CanUnit :="";
boPin157.Description :="for the Neotec diag pages";
boPin157.ErrorReaction := eErrorReaction.ERSIG_DFLT;
boPin157.ReceiverAdress :=1;
boPin157.ToolScalingDivisor :=1;
boPin157.ToolScalingMultiplier :=1;
boPin157.ToolScalingOffset :=0;
boPin157.ToolUnit :="";

boPin181.AppScalingDivisor :=1;
boPin181.AppScalingMultiplier :=1;
boPin181.AppScalingOffset :=0;
boPin181.AppUnit :="";
boPin181.CanDefault :=0;
boPin181.CanInit :=0;
boPin181.CanMax :=1;
boPin181.CanMin :=0;
boPin181.CanUnit :="";
boPin181.Description :="for the Neotec diag pages";
boPin181.ErrorReaction := eErrorReaction.ERSIG_DFLT;
boPin181.ReceiverAdress :=1;
boPin181.ToolScalingDivisor :=1;
boPin181.ToolScalingMultiplier :=1;
boPin181.ToolScalingOffset :=0;
boPin181.ToolUnit :="";

boPin160.AppScalingDivisor :=1;
boPin160.AppScalingMultiplier :=1;
boPin160.AppScalingOffset :=0;
boPin160.AppUnit :="";
boPin160.CanDefault :=0;
boPin160.CanInit :=0;
boPin160.CanMax :=1;
boPin160.CanMin :=0;
boPin160.CanUnit :="";
boPin160.Description :="for the Neotec diag pages";
boPin160.ErrorReaction := eErrorReaction.ERSIG_DFLT;
boPin160.ReceiverAdress :=1;
boPin160.ToolScalingDivisor :=1;
boPin160.ToolScalingMultiplier :=1;
boPin160.ToolScalingOffset :=0;
boPin160.ToolUnit :="";

boPin184.AppScalingDivisor :=1;
boPin184.AppScalingMultiplier :=1;
boPin184.AppScalingOffset :=0;
boPin184.AppUnit :="";
boPin184.CanDefault :=0;
boPin184.CanInit :=0;
boPin184.CanMax :=1;
boPin184.CanMin :=0;
boPin184.CanUnit :="";
boPin184.Description :="for the Neotec diag pages";
boPin184.ErrorReaction := eErrorReaction.ERSIG_DFLT;
boPin184.ReceiverAdress :=1;
boPin184.ToolScalingDivisor :=1;
boPin184.ToolScalingMultiplier :=1;
boPin184.ToolScalingOffset :=0;
boPin184.ToolUnit :="";

boPin187.AppScalingDivisor :=1;
boPin187.AppScalingMultiplier :=1;
boPin187.AppScalingOffset :=0;
boPin187.AppUnit :="";
boPin187.CanDefault :=0;
boPin187.CanInit :=0;
boPin187.CanMax :=1;
boPin187.CanMin :=0;
boPin187.CanUnit :="";
boPin187.Description :="for the Neotec diag pages";
boPin187.ErrorReaction := eErrorReaction.ERSIG_DFLT;
boPin187.ReceiverAdress :=1;
boPin187.ToolScalingDivisor :=1;
boPin187.ToolScalingMultiplier :=1;
boPin187.ToolScalingOffset :=0;
boPin187.ToolUnit :="";

boPin163.AppScalingDivisor :=1;
boPin163.AppScalingMultiplier :=1;
boPin163.AppScalingOffset :=0;
boPin163.AppUnit :="";
boPin163.CanDefault :=0;
boPin163.CanInit :=0;
boPin163.CanMax :=1;
boPin163.CanMin :=0;
boPin163.CanUnit :="";
boPin163.Description :="for the Neotec diag pages";
boPin163.ErrorReaction := eErrorReaction.ERSIG_DFLT;
boPin163.ReceiverAdress :=1;
boPin163.ToolScalingDivisor :=1;
boPin163.ToolScalingMultiplier :=1;
boPin163.ToolScalingOffset :=0;
boPin163.ToolUnit :="";

boPin149.AppScalingDivisor :=1;
boPin149.AppScalingMultiplier :=1;
boPin149.AppScalingOffset :=0;
boPin149.AppUnit :="";
boPin149.CanDefault :=0;
boPin149.CanInit :=0;
boPin149.CanMax :=1;
boPin149.CanMin :=0;
boPin149.CanUnit :="";
boPin149.Description :="for the Neotec diag pages";
boPin149.ErrorReaction := eErrorReaction.ERSIG_DFLT;
boPin149.ReceiverAdress :=1;
boPin149.ToolScalingDivisor :=1;
boPin149.ToolScalingMultiplier :=1;
boPin149.ToolScalingOffset :=0;
boPin149.ToolUnit :="";

boPin173.AppScalingDivisor :=1;
boPin173.AppScalingMultiplier :=1;
boPin173.AppScalingOffset :=0;
boPin173.AppUnit :="";
boPin173.CanDefault :=0;
boPin173.CanInit :=0;
boPin173.CanMax :=1;
boPin173.CanMin :=0;
boPin173.CanUnit :="";
boPin173.Description :="for the Neotec diag pages";
boPin173.ErrorReaction := eErrorReaction.ERSIG_DFLT;
boPin173.ReceiverAdress :=1;
boPin173.ToolScalingDivisor :=1;
boPin173.ToolScalingMultiplier :=1;
boPin173.ToolScalingOffset :=0;
boPin173.ToolUnit :="";

boPin152.AppScalingDivisor :=1;
boPin152.AppScalingMultiplier :=1;
boPin152.AppScalingOffset :=0;
boPin152.AppUnit :="";
boPin152.CanDefault :=0;
boPin152.CanInit :=0;
boPin152.CanMax :=1;
boPin152.CanMin :=0;
boPin152.CanUnit :="";
boPin152.Description :="for the Neotec diag pages";
boPin152.ErrorReaction := eErrorReaction.ERSIG_DFLT;
boPin152.ReceiverAdress :=1;
boPin152.ToolScalingDivisor :=1;
boPin152.ToolScalingMultiplier :=1;
boPin152.ToolScalingOffset :=0;
boPin152.ToolUnit :="";

boPin176.AppScalingDivisor :=1;
boPin176.AppScalingMultiplier :=1;
boPin176.AppScalingOffset :=0;
boPin176.AppUnit :="";
boPin176.CanDefault :=0;
boPin176.CanInit :=0;
boPin176.CanMax :=1;
boPin176.CanMin :=0;
boPin176.CanUnit :="";
boPin176.Description :="for the Neotec diag pages";
boPin176.ErrorReaction := eErrorReaction.ERSIG_DFLT;
boPin176.ReceiverAdress :=1;
boPin176.ToolScalingDivisor :=1;
boPin176.ToolScalingMultiplier :=1;
boPin176.ToolScalingOffset :=0;
boPin176.ToolUnit :="";

boPin155.AppScalingDivisor :=1;
boPin155.AppScalingMultiplier :=1;
boPin155.AppScalingOffset :=0;
boPin155.AppUnit :="";
boPin155.CanDefault :=0;
boPin155.CanInit :=0;
boPin155.CanMax :=1;
boPin155.CanMin :=0;
boPin155.CanUnit :="";
boPin155.Description :="for the Neotec diag pages";
boPin155.ErrorReaction := eErrorReaction.ERSIG_DFLT;
boPin155.ReceiverAdress :=1;
boPin155.ToolScalingDivisor :=1;
boPin155.ToolScalingMultiplier :=1;
boPin155.ToolScalingOffset :=0;
boPin155.ToolUnit :="";

boPin179.AppScalingDivisor :=1;
boPin179.AppScalingMultiplier :=1;
boPin179.AppScalingOffset :=0;
boPin179.AppUnit :="";
boPin179.CanDefault :=0;
boPin179.CanInit :=0;
boPin179.CanMax :=1;
boPin179.CanMin :=0;
boPin179.CanUnit :="";
boPin179.Description :="for the Neotec diag pages";
boPin179.ErrorReaction := eErrorReaction.ERSIG_DFLT;
boPin179.ReceiverAdress :=1;
boPin179.ToolScalingDivisor :=1;
boPin179.ToolScalingMultiplier :=1;
boPin179.ToolScalingOffset :=0;
boPin179.ToolUnit :="";

boPin158.AppScalingDivisor :=1;
boPin158.AppScalingMultiplier :=1;
boPin158.AppScalingOffset :=0;
boPin158.AppUnit :="";
boPin158.CanDefault :=0;
boPin158.CanInit :=0;
boPin158.CanMax :=1;
boPin158.CanMin :=0;
boPin158.CanUnit :="";
boPin158.Description :="for the Neotec diag pages";
boPin158.ErrorReaction := eErrorReaction.ERSIG_DFLT;
boPin158.ReceiverAdress :=1;
boPin158.ToolScalingDivisor :=1;
boPin158.ToolScalingMultiplier :=1;
boPin158.ToolScalingOffset :=0;
boPin158.ToolUnit :="";

boPin182.AppScalingDivisor :=1;
boPin182.AppScalingMultiplier :=1;
boPin182.AppScalingOffset :=0;
boPin182.AppUnit :="";
boPin182.CanDefault :=0;
boPin182.CanInit :=0;
boPin182.CanMax :=1;
boPin182.CanMin :=0;
boPin182.CanUnit :="";
boPin182.Description :="for the Neotec diag pages";
boPin182.ErrorReaction := eErrorReaction.ERSIG_DFLT;
boPin182.ReceiverAdress :=1;
boPin182.ToolScalingDivisor :=1;
boPin182.ToolScalingMultiplier :=1;
boPin182.ToolScalingOffset :=0;
boPin182.ToolUnit :="";

boPin251.AppScalingDivisor :=1;
boPin251.AppScalingMultiplier :=1;
boPin251.AppScalingOffset :=0;
boPin251.AppUnit :="";
boPin251.CanDefault :=0;
boPin251.CanInit :=0;
boPin251.CanMax :=1;
boPin251.CanMin :=0;
boPin251.CanUnit :="";
boPin251.Description :="for the Neotec diag pages";
boPin251.ErrorReaction := eErrorReaction.ERSIG_DFLT;
boPin251.ReceiverAdress :=1;
boPin251.ToolScalingDivisor :=1;
boPin251.ToolScalingMultiplier :=1;
boPin251.ToolScalingOffset :=0;
boPin251.ToolUnit :="";

boPin186.AppScalingDivisor :=1;
boPin186.AppScalingMultiplier :=1;
boPin186.AppScalingOffset :=0;
boPin186.AppUnit :="";
boPin186.CanDefault :=0;
boPin186.CanInit :=0;
boPin186.CanMax :=1;
boPin186.CanMin :=0;
boPin186.CanUnit :="";
boPin186.Description :="for the Neotec diag pages";
boPin186.ErrorReaction := eErrorReaction.ERSIG_DFLT;
boPin186.ReceiverAdress :=1;
boPin186.ToolScalingDivisor :=1;
boPin186.ToolScalingMultiplier :=1;
boPin186.ToolScalingOffset :=0;
boPin186.ToolUnit :="";

boPin239.AppScalingDivisor :=1;
boPin239.AppScalingMultiplier :=1;
boPin239.AppScalingOffset :=0;
boPin239.AppUnit :="";
boPin239.CanDefault :=0;
boPin239.CanInit :=0;
boPin239.CanMax :=1;
boPin239.CanMin :=0;
boPin239.CanUnit :="";
boPin239.Description :="for the Neotec diag pages";
boPin239.ErrorReaction := eErrorReaction.ERSIG_DFLT;
boPin239.ReceiverAdress :=1;
boPin239.ToolScalingDivisor :=1;
boPin239.ToolScalingMultiplier :=1;
boPin239.ToolScalingOffset :=0;
boPin239.ToolUnit :="";


                
END_METHOD
END_FUNCTION_BLOCK

FUNCTION_BLOCK Msg6C1SendToEvision7MessageClass EXTENDS CanReceiveMessageClass
  VAR_INPUT
    boPin230Fault : BoolCanSignalClass;
    boPin243Fault : BoolCanSignalClass;
    boPin244Fault : BoolCanSignalClass;
    boPin245Fault : BoolCanSignalClass;
    boPin256Fault : BoolCanSignalClass;
    boPin257Fault : BoolCanSignalClass;
    boPin258Fault : BoolCanSignalClass;
    boPin103Fault : BoolCanSignalClass;
    boPin127Fault : BoolCanSignalClass;
    boPin104Fault : BoolCanSignalClass;
    boPin128Fault : BoolCanSignalClass;
    boPin105Fault : BoolCanSignalClass;
    boPin129Fault : BoolCanSignalClass;
    boPin106Fault : BoolCanSignalClass;
    boPin130Fault : BoolCanSignalClass;
    boPin107Fault : BoolCanSignalClass;
    boPin131Fault : BoolCanSignalClass;
    boPin108Fault : BoolCanSignalClass;
    boPin132Fault : BoolCanSignalClass;
    boPin109Fault : BoolCanSignalClass;
    boPin133Fault : BoolCanSignalClass;
    boPin110Fault : BoolCanSignalClass;
    boPin134Fault : BoolCanSignalClass;
    boPin111Fault : BoolCanSignalClass;
    boPin135Fault : BoolCanSignalClass;
    boPin112Fault : BoolCanSignalClass;
    boPin136Fault : BoolCanSignalClass;
    boPin113Fault : BoolCanSignalClass;
    boPin137Fault : BoolCanSignalClass;
    boPin114Fault : BoolCanSignalClass;
    boPin138Fault : BoolCanSignalClass;
    boPin115Fault : BoolCanSignalClass;
    boPin139Fault : BoolCanSignalClass;
    boPin116Fault : BoolCanSignalClass;
    boPin140Fault : BoolCanSignalClass;
    boPin117Fault : BoolCanSignalClass;
    boPin141Fault : BoolCanSignalClass;
    boPin122Fault : BoolCanSignalClass;
    boPin146Fault : BoolCanSignalClass;
    boPin123Fault : BoolCanSignalClass;
    boPin147Fault : BoolCanSignalClass;
    boPin124Fault : BoolCanSignalClass;
    boPin148Fault : BoolCanSignalClass;
    boPin153Fault : BoolCanSignalClass;
    boPin177Fault : BoolCanSignalClass;
    boPin156Fault : BoolCanSignalClass;
    boPin180Fault : BoolCanSignalClass;
    boPin159Fault : BoolCanSignalClass;
    boPin183Fault : BoolCanSignalClass;
    boPin186Fault : BoolCanSignalClass;
    boPin162Fault : BoolCanSignalClass;
    boPin189Fault : BoolCanSignalClass;
    boPin165Fault : BoolCanSignalClass;
    boPin192Fault : BoolCanSignalClass;
    boPin168Fault : BoolCanSignalClass;
    boPin195Fault : BoolCanSignalClass;
    boPin171Fault : BoolCanSignalClass;
    boPin154Fault : BoolCanSignalClass;
    boPin178Fault : BoolCanSignalClass;
    boPin157Fault : BoolCanSignalClass;
    boPin181Fault : BoolCanSignalClass;
    boPin160Fault : BoolCanSignalClass;
    boPin184Fault : BoolCanSignalClass;
    boPin187Fault : BoolCanSignalClass;
    Counter : UInt32CanSignalClass;
  END_VAR

            
          

METHOD SetData
  VAR_INPUT
    CanMsgPointer : POINTER TO CanMessageClass;
  END_VAR
                  IF IsValidPointer(canMsgPointer,'SetData') THEN
	SUPER^.SetData(CanMsgPointer);
	//Set the new data
	boPin230Fault.Value := canMsgPointer^.GetBoolOnBit(0);
	boPin243Fault.Value := canMsgPointer^.GetBoolOnBit(1);
	boPin244Fault.Value := canMsgPointer^.GetBoolOnBit(2);
	boPin245Fault.Value := canMsgPointer^.GetBoolOnBit(3);
	boPin256Fault.Value := canMsgPointer^.GetBoolOnBit(4);
	boPin257Fault.Value := canMsgPointer^.GetBoolOnBit(5);
	boPin258Fault.Value := canMsgPointer^.GetBoolOnBit(6);
	boPin103Fault.Value := canMsgPointer^.GetBoolOnBit(7);
	boPin127Fault.Value := canMsgPointer^.GetBoolOnBit(8);
	boPin104Fault.Value := canMsgPointer^.GetBoolOnBit(9);
	boPin128Fault.Value := canMsgPointer^.GetBoolOnBit(10);
	boPin105Fault.Value := canMsgPointer^.GetBoolOnBit(11);
	boPin129Fault.Value := canMsgPointer^.GetBoolOnBit(12);
	boPin106Fault.Value := canMsgPointer^.GetBoolOnBit(13);
	boPin130Fault.Value := canMsgPointer^.GetBoolOnBit(14);
	boPin107Fault.Value := canMsgPointer^.GetBoolOnBit(15);
	boPin131Fault.Value := canMsgPointer^.GetBoolOnBit(16);
	boPin108Fault.Value := canMsgPointer^.GetBoolOnBit(17);
	boPin132Fault.Value := canMsgPointer^.GetBoolOnBit(18);
	boPin109Fault.Value := canMsgPointer^.GetBoolOnBit(19);
	boPin133Fault.Value := canMsgPointer^.GetBoolOnBit(20);
	boPin110Fault.Value := canMsgPointer^.GetBoolOnBit(21);
	boPin134Fault.Value := canMsgPointer^.GetBoolOnBit(22);
	boPin111Fault.Value := canMsgPointer^.GetBoolOnBit(23);
	boPin135Fault.Value := canMsgPointer^.GetBoolOnBit(24);
	boPin112Fault.Value := canMsgPointer^.GetBoolOnBit(25);
	boPin136Fault.Value := canMsgPointer^.GetBoolOnBit(26);
	boPin113Fault.Value := canMsgPointer^.GetBoolOnBit(27);
	boPin137Fault.Value := canMsgPointer^.GetBoolOnBit(28);
	boPin114Fault.Value := canMsgPointer^.GetBoolOnBit(29);
	boPin138Fault.Value := canMsgPointer^.GetBoolOnBit(30);
	boPin115Fault.Value := canMsgPointer^.GetBoolOnBit(31);
	boPin139Fault.Value := canMsgPointer^.GetBoolOnBit(32);
	boPin116Fault.Value := canMsgPointer^.GetBoolOnBit(33);
	boPin140Fault.Value := canMsgPointer^.GetBoolOnBit(34);
	boPin117Fault.Value := canMsgPointer^.GetBoolOnBit(35);
	boPin141Fault.Value := canMsgPointer^.GetBoolOnBit(36);
	boPin122Fault.Value := canMsgPointer^.GetBoolOnBit(37);
	boPin146Fault.Value := canMsgPointer^.GetBoolOnBit(38);
	boPin123Fault.Value := canMsgPointer^.GetBoolOnBit(39);
	boPin147Fault.Value := canMsgPointer^.GetBoolOnBit(40);
	boPin124Fault.Value := canMsgPointer^.GetBoolOnBit(41);
	boPin148Fault.Value := canMsgPointer^.GetBoolOnBit(42);
	boPin153Fault.Value := canMsgPointer^.GetBoolOnBit(43);
	boPin177Fault.Value := canMsgPointer^.GetBoolOnBit(44);
	boPin156Fault.Value := canMsgPointer^.GetBoolOnBit(45);
	boPin180Fault.Value := canMsgPointer^.GetBoolOnBit(46);
	boPin159Fault.Value := canMsgPointer^.GetBoolOnBit(47);
	boPin183Fault.Value := canMsgPointer^.GetBoolOnBit(48);
	boPin186Fault.Value := canMsgPointer^.GetBoolOnBit(49);
	boPin162Fault.Value := canMsgPointer^.GetBoolOnBit(50);
	boPin189Fault.Value := canMsgPointer^.GetBoolOnBit(51);
	boPin165Fault.Value := canMsgPointer^.GetBoolOnBit(52);
	boPin192Fault.Value := canMsgPointer^.GetBoolOnBit(53);
	boPin168Fault.Value := canMsgPointer^.GetBoolOnBit(54);
	boPin195Fault.Value := canMsgPointer^.GetBoolOnBit(55);
	boPin171Fault.Value := canMsgPointer^.GetBoolOnBit(56);
	boPin154Fault.Value := canMsgPointer^.GetBoolOnBit(57);
	boPin178Fault.Value := canMsgPointer^.GetBoolOnBit(58);
	boPin157Fault.Value := canMsgPointer^.GetBoolOnBit(59);
	boPin181Fault.Value := canMsgPointer^.GetBoolOnBit(60);
	boPin160Fault.Value := canMsgPointer^.GetBoolOnBit(61);
	boPin184Fault.Value := canMsgPointer^.GetBoolOnBit(62);
	boPin187Fault.Value := canMsgPointer^.GetBoolOnBit(63);
	//And increase the counter
	Counter.Value := CanMsgPointer^.Counter.Value;
END_IF

                
END_METHOD

PROPERTY boPin230FaultRawValue : BOOL
GET
                    boPin230FaultRawValue := boPin230Fault.Value;

                  
END_GET
END_PROPERTY

PROPERTY boPin243FaultRawValue : BOOL
GET
                    boPin243FaultRawValue := boPin243Fault.Value;

                  
END_GET
END_PROPERTY

PROPERTY boPin244FaultRawValue : BOOL
GET
                    boPin244FaultRawValue := boPin244Fault.Value;

                  
END_GET
END_PROPERTY

PROPERTY boPin245FaultRawValue : BOOL
GET
                    boPin245FaultRawValue := boPin245Fault.Value;

                  
END_GET
END_PROPERTY

PROPERTY boPin256FaultRawValue : BOOL
GET
                    boPin256FaultRawValue := boPin256Fault.Value;

                  
END_GET
END_PROPERTY

PROPERTY boPin257FaultRawValue : BOOL
GET
                    boPin257FaultRawValue := boPin257Fault.Value;

                  
END_GET
END_PROPERTY

PROPERTY boPin258FaultRawValue : BOOL
GET
                    boPin258FaultRawValue := boPin258Fault.Value;

                  
END_GET
END_PROPERTY

PROPERTY boPin103FaultRawValue : BOOL
GET
                    boPin103FaultRawValue := boPin103Fault.Value;

                  
END_GET
END_PROPERTY

PROPERTY boPin127FaultRawValue : BOOL
GET
                    boPin127FaultRawValue := boPin127Fault.Value;

                  
END_GET
END_PROPERTY

PROPERTY boPin104FaultRawValue : BOOL
GET
                    boPin104FaultRawValue := boPin104Fault.Value;

                  
END_GET
END_PROPERTY

